LIN {X 0,Y 117.45,Z 837.122,A -85,B 0,C 180,E1 28506.231,E2 28506.231} C_VEL
LIN {X 0,Y 123.692,Z 839.313,A -85,B 0,C 180,E1 28517.447,E2 28517.447} C_VEL
LIN {X 0,Y 126.068,Z 840.042,A -85,B 0,C 180,E1 28523.129,E2 28523.129} C_VEL
LIN {X 0,Y 128.758,Z 840.316,A -85,B 0,C 180,E1 28530.003,E2 28530.003} C_VEL
LIN {X 0,Y 126.025,Z 840.042,A -85,B 0,C 180,E1 28536.88,E2 28536.88} C_VEL
LIN {X 0,Y 122.693,Z 839.07,A -85,B 0,C 180,E1 28544.243,E2 28544.243} C_VEL
LIN {X 0,Y 118.511,Z 837.415,A -85,B 0,C 180,E1 28552.461,E2 28552.461} C_VEL
LIN {X 0,Y 109.257,Z 835.091,A -85,B 0,C 180,E1 28564.022,E2 28564.022} C_VEL
LIN {X 0,Y 99.295,Z 832.926,A -85,B 0,C 180,E1 28577.915,E2 28577.915} C_VEL
LIN {X 0,Y 67.915,Z 840.094,A -85,B 0,C 180,E1 28563.751,E2 28563.751} C_VEL
LIN {X 0,Y 48.693,Z 842.803,A -85,B 0,C 180,E1 28530.008,E2 28530.008} C_VEL
LIN {X 0,Y 67.859,Z 840.097,A -85,B 0,C 180,E1 28496.232,E2 28496.232} C_VEL
LIN {X 0,Y 93.632,Z 834.401,A -85,B 0,C 180,E1 28483.517,E2 28483.517} C_VEL
LIN {X 0,Y 99.85,Z 833.009,A -85,B 0,C 180,E1 28482.861,E2 28482.861} C_VEL
LIN {X 0,Y 109.786,Z 835.227,A -85,B 0,C 180,E1 28496.651,E2 28496.651} C_VEL
LIN {X 0,Y 117.45,Z 837.122,A -85,B 0,C 180,E1 28506.231,E2 28506.231} C_VEL
LIN {X 0,Y 119.061,Z 838.09,A -85,B 0,C 180,E1 28510.313,E2 28510.313} C_VEL
LIN {X 0,Y 117.917,Z 840.331,A -85,B 0,C 180,E1 28523.404,E2 28523.404} C_VEL
LIN {X 0,Y 120.645,Z 840.568,A -85,B 0,C 180,E1 28530.003,E2 28530.003} C_VEL
LIN {X 0,Y 117.661,Z 840.304,A -85,B 0,C 180,E1 28537.372,E2 28537.372} C_VEL
LIN {X 0,Y 111.816,Z 838.693,A -85,B 0,C 180,E1 28549.125,E2 28549.125} C_VEL
LIN {X 0,Y 107.871,Z 837.778,A -85,B 0,C 180,E1 28554.818,E2 28554.818} C_VEL
LIN {X 0,Y 95.953,Z 835.393,A -85,B 0,C 180,E1 28570.441,E2 28570.441} C_VEL
LIN {X 0,Y 92.882,Z 835.886,A -85,B 0,C 180,E1 28570.537,E2 28570.537} C_VEL
LIN {X 0,Y 63.467,Z 841.732,A -85,B 0,C 180,E1 28547.957,E2 28547.957} C_VEL
LIN {X 0,Y 56.707,Z 842.554,A -85,B 0,C 180,E1 28530.007,E2 28530.007} C_VEL
LIN {X 0,Y 74.763,Z 839.843,A -85,B 0,C 180,E1 28499.702,E2 28499.702} C_VEL
LIN {X 0,Y 92.876,Z 835.889,A -85,B 0,C 180,E1 28489.471,E2 28489.471} C_VEL
LIN {X 0,Y 95.998,Z 835.377,A -85,B 0,C 180,E1 28489.529,E2 28489.529} C_VEL
LIN {X 0,Y 107.958,Z 837.777,A -85,B 0,C 180,E1 28505.212,E2 28505.212} C_VEL
LIN {X 0,Y 111.852,Z 838.68,A -85,B 0,C 180,E1 28510.823,E2 28510.823} C_VEL
LIN {X 0,Y 117.917,Z 840.331,A -85,B 0,C 180,E1 28523.404,E2 28523.404} C_VEL
LIN {X 0,Y 116.337,Z 840.614,A -85,B 0,C 180,E1 28527.551,E2 28527.551} C_VEL
LIN {X 0,Y 110.179,Z 840.674,A -85,B 0,C 180,E1 28534.68,E2 28534.68} C_VEL
LIN {X 0,Y 107.551,Z 840.278,A -85,B 0,C 180,E1 28540.803,E2 28540.803} C_VEL
LIN {X 0,Y 104.839,Z 839.648,A -85,B 0,C 180,E1 28546.735,E2 28546.735} C_VEL
LIN {X 0,Y 96.704,Z 838.168,A -85,B 0,C 180,E1 28557.918,E2 28557.918} C_VEL
LIN {X 0,Y 92.654,Z 837.576,A -85,B 0,C 180,E1 28562.71,E2 28562.71} C_VEL
LIN {X 0,Y 89.467,Z 838.001,A -85,B 0,C 180,E1 28562.489,E2 28562.489} C_VEL
LIN {X 0,Y 69.132,Z 841.835,A -85,B 0,C 180,E1 28542.614,E2 28542.614} C_VEL
LIN {X 0,Y 64.726,Z 842.305,A -85,B 0,C 180,E1 28530.006,E2 28530.006} C_VEL
LIN {X 0,Y 81.92,Z 839.588,A -85,B 0,C 180,E1 28502.585,E2 28502.585} C_VEL
LIN {X 0,Y 89.524,Z 837.982,A -85,B 0,C 180,E1 28497.454,E2 28497.454} C_VEL
LIN {X 0,Y 92.693,Z 837.57,A -85,B 0,C 180,E1 28497.288,E2 28497.288} C_VEL
LIN {X 0,Y 99.504,Z 838.587,A -85,B 0,C 180,E1 28505.514,E2 28505.514} C_VEL
LIN {X 0,Y 104.9,Z 839.648,A -85,B 0,C 180,E1 28513.283,E2 28513.283} C_VEL
LIN {X 0,Y 109.758,Z 840.638,A -85,B 0,C 180,E1 28524.137,E2 28524.137} C_VEL
LIN {X 0,Y 112.484,Z 840.821,A -85,B 0,C 180,E1 28530.004,E2 28530.004} C_VEL
LIN {X 0,Y 110.179,Z 840.674,A -85,B 0,C 180,E1 28534.68,E2 28534.68} C_VEL
LIN {X 0,Y 105.682,Z 840.634,A -85,B 0,C 180,E1 28538.598,E2 28538.598} C_VEL
LIN {X 0,Y 96.395,Z 840.259,A -85,B 0,C 180,E1 28545.328,E2 28545.328} C_VEL
LIN {X 0,Y 90.521,Z 839.276,A -85,B 0,C 180,E1 28554.711,E2 28554.711} C_VEL
LIN {X 0,Y 84.585,Z 840.315,A -85,B 0,C 180,E1 28550.909,E2 28550.909} C_VEL
LIN {X 0,Y 72.751,Z 842.055,A -85,B 0,C 180,E1 28530.006,E2 28530.006} C_VEL
LIN {X 0,Y 84.537,Z 840.318,A -85,B 0,C 180,E1 28509.089,E2 28509.089} C_VEL
LIN {X 0,Y 90.571,Z 839.27,A -85,B 0,C 180,E1 28505.276,E2 28505.276} C_VEL
LIN {X 0,Y 95.229,Z 840.033,A -85,B 0,C 180,E1 28511.974,E2 28511.974} C_VEL
LIN {X 0,Y 100.503,Z 840.844,A -85,B 0,C 180,E1 28521.369,E2 28521.369} C_VEL
LIN {X 0,Y 104.257,Z 841.077,A -85,B 0,C 180,E1 28530.004,E2 28530.004} C_VEL
LIN {X 0,Y 100.458,Z 840.844,A -85,B 0,C 180,E1 28538.643,E2 28538.643} C_VEL
LIN {X 0,Y 96.395,Z 840.259,A -85,B 0,C 180,E1 28545.328,E2 28545.328} C_VEL
LIN {X 0,Y 92.31,Z 840.489,A -85,B 0,C 180,E1 28545.322,E2 28545.322} C_VEL
LIN {X 0,Y 86.505,Z 841.177,A -85,B 0,C 180,E1 28541.158,E2 28541.158} C_VEL
LIN {X 0,Y 81.835,Z 841.654,A -85,B 0,C 180,E1 28533.397,E2 28533.397} C_VEL
LIN {X 0,Y 80.762,Z 841.807,A -85,B 0,C 180,E1 28530.005,E2 28530.005} C_VEL
LIN {X 0,Y 88.556,Z 840.741,A -85,B 0,C 180,E1 28515.404,E2 28515.404} C_VEL
LIN {X 0,Y 91.692,Z 841.15,A -85,B 0,C 180,E1 28520.966,E2 28520.966} C_VEL
LIN {X 0,Y 95.951,Z 841.335,A -85,B 0,C 180,E1 28530.004,E2 28530.004} C_VEL
LIN {X 0,Y 91.361,Z 841.131,A -85,B 0,C 180,E1 28539.512,E2 28539.512} C_VEL
LIN {X 0,Y 88.558,Z 840.746,A -85,B 0,C 180,E1 28544.541,E2 28544.541} C_VEL
LIN {X 0,Y 81.835,Z 841.654,A -85,B 0,C 180,E1 28533.397,E2 28533.397} C_VEL
LIN {X 0,Y 81.379,Z 843.653,A -85,B 0,C 180,E1 28532.075,E2 28532.075} C_VEL
LIN {X 0,Y 81.379,Z 862.5,A -85,B 0,C 180,E1 28532.075,E2 28532.075} C_VEL
LIN {X 0,Y 81.379,Z 862.5,A -85,B 0,C 180,E1 28532.075,E2 28532.075}

QRS_NEXT_CUT()
PTP {E1 28616.872,E2 28616.872}
PTP {X 0,Y 607.922,A -85,B 0,C 180,E1 28616.872,E2 28616.872,E3 0,E4 0,E5 0,E6 0}
QRS_SPEED_INIT()
LIN {X 0,Y 607.922,Z 862.5,A -85,B 0,C 180,E1 28616.872,E2 28616.872,E3 0,E4 0,E5 0,E6 0} C_VEL
LIN {X 0,Y 607.922,Z 274.59,A -85,B 0,C 180,E1 28616.872,E2 28616.872} C_VEL
LIN {X 0,Y 607.922,Z 266.51,A -85,B 0,C 180,E1 28616.872,E2 28616.872} C_VEL
LIN {X 0,Y 607.915,Z 264.51,A -85,B 0,C 180,E1 28616.683,E2 28616.683} C_VEL
LIN {X 0,Y 607.865,Z 264.511,A -85,B 0,C 180,E1 28613.578,E2 28613.578} C_VEL
LIN {X 0,Y 607.916,Z 264.507,A -85,B 0,C 180,E1 28610.438,E2 28610.438} C_VEL
LIN {X 0,Y 607.87,Z 264.512,A -85,B 0,C 180,E1 28607.363,E2 28607.363} C_VEL
LIN {X 0,Y 607.908,Z 264.506,A -85,B 0,C 180,E1 28604.155,E2 28604.155} C_VEL
LIN {X 0,Y 607.891,Z 264.513,A -85,B 0,C 180,E1 28600.994,E2 28600.994} C_VEL
LIN {X 0,Y 607.884,Z 264.508,A -85,B 0,C 180,E1 28597.771,E2 28597.771} C_VEL
LIN {X 0,Y 607.913,Z 264.516,A -85,B 0,C 180,E1 28594.683,E2 28594.683} C_VEL
LIN {X 0,Y 607.876,Z 264.509,A -85,B 0,C 180,E1 28591.44,E2 28591.44} C_VEL
LIN {X 0,Y 607.911,Z 264.511,A -85,B 0,C 180,E1 28588.354,E2 28588.354} C_VEL
LIN {X 0,Y 607.877,Z 264.509,A -85,B 0,C 180,E1 28585.312,E2 28585.312} C_VEL
LIN {X 0,Y 607.909,Z 264.511,A -85,B 0,C 180,E1 28582.277,E2 28582.277} C_VEL
LIN {X 0,Y 607.879,Z 264.51,A -85,B 0,C 180,E1 28579.165,E2 28579.165} C_VEL
LIN {X 0,Y 607.908,Z 264.508,A -85,B 0,C 180,E1 28576.046,E2 28576.046} C_VEL
LIN {X 0,Y 607.884,Z 264.511,A -85,B 0,C 180,E1 28572.917,E2 28572.917} C_VEL
LIN {X 0,Y 607.913,Z 264.506,A -85,B 0,C 180,E1 28569.776,E2 28569.776} C_VEL
LIN {X 0,Y 607.904,Z 264.514,A -85,B 0,C 180,E1 28566.54,E2 28566.54} C_VEL
LIN {X 0,Y 607.898,Z 264.506,A -85,B 0,C 180,E1 28563.322,E2 28563.322} C_VEL
LIN {X 0,Y 607.908,Z 264.512,A -85,B 0,C 180,E1 28560.102,E2 28560.102} C_VEL
LIN {X 0,Y 607.888,Z 264.508,A -85,B 0,C 180,E1 28556.94,E2 28556.94} C_VEL
LIN {X 0,Y 607.903,Z 264.508,A -85,B 0,C 180,E1 28553.763,E2 28553.763} C_VEL
LIN {X 0,Y 607.892,Z 264.511,A -85,B 0,C 180,E1 28550.628,E2 28550.628} C_VEL
LIN {X 0,Y 607.911,Z 264.505,A -85,B 0,C 180,E1 28547.418,E2 28547.418} C_VEL
LIN {X 0,Y 607.915,Z 264.514,A -85,B 0,C 180,E1 28544.088,E2 28544.088} C_VEL
LIN {X 0,Y 607.899,Z 264.506,A -85,B 0,C 180,E1 28540.903,E2 28540.903} C_VEL
LIN {X 0,Y 607.9,Z 264.511,A -85,B 0,C 180,E1 28537.751,E2 28537.751} C_VEL
LIN {X 0,Y 607.895,Z 264.508,A -85,B 0,C 180,E1 28534.623,E2 28534.623} C_VEL
LIN {X 0,Y 607.897,Z 264.509,A -85,B 0,C 180,E1 28531.508,E2 28531.508} C_VEL
LIN {X 0,Y 607.897,Z 264.51,A -85,B 0,C 180,E1 28528.398,E2 28528.398} C_VEL
LIN {X 0,Y 607.9,Z 264.506,A -85,B 0,C 180,E1 28525.188,E2 28525.188} C_VEL
LIN {X 0,Y 607.911,Z 264.515,A -85,B 0,C 180,E1 28521.944,E2 28521.944} C_VEL
LIN {X 0,Y 607.912,Z 264.505,A -85,B 0,C 180,E1 28518.713,E2 28518.713} C_VEL
LIN {X 0,Y 607.896,Z 264.512,A -85,B 0,C 180,E1 28515.522,E2 28515.522} C_VEL
LIN {X 0,Y 607.903,Z 264.508,A -85,B 0,C 180,E1 28512.384,E2 28512.384} C_VEL
LIN {X 0,Y 607.89,Z 264.51,A -85,B 0,C 180,E1 28509.291,E2 28509.291} C_VEL
LIN {X 0,Y 607.903,Z 264.508,A -85,B 0,C 180,E1 28506.237,E2 28506.237} C_VEL
LIN {X 0,Y 607.888,Z 264.508,A -85,B 0,C 180,E1 28503.06,E2 28503.06} C_VEL
LIN {X 0,Y 607.908,Z 264.512,A -85,B 0,C 180,E1 28499.892,E2 28499.892} C_VEL
LIN {X 0,Y 607.899,Z 264.506,A -85,B 0,C 180,E1 28496.673,E2 28496.673} C_VEL
LIN {X 0,Y 607.895,Z 264.512,A -85,B 0,C 180,E1 28493.342,E2 28493.342} C_VEL
LIN {X 0,Y 607.911,Z 264.506,A -85,B 0,C 180,E1 28490.183,E2 28490.183} C_VEL
LIN {X 0,Y 607.883,Z 264.511,A -85,B 0,C 180,E1 28487.049,E2 28487.049} C_VEL
LIN {X 0,Y 607.908,Z 264.509,A -85,B 0,C 180,E1 28483.914,E2 28483.914} C_VEL
LIN {X 0,Y 607.88,Z 264.509,A -85,B 0,C 180,E1 28480.768,E2 28480.768} C_VEL
LIN {X 0,Y 607.911,Z 264.513,A -85,B 0,C 180,E1 28477.604,E2 28477.604} C_VEL
LIN {X 0,Y 607.885,Z 264.508,A -85,B 0,C 180,E1 28474.459,E2 28474.459} C_VEL
LIN {X 0,Y 607.9,Z 264.514,A -85,B 0,C 180,E1 28471.205,E2 28471.205} C_VEL
LIN {X 0,Y 607.913,Z 264.506,A -85,B 0,C 180,E1 28467.969,E2 28467.969} C_VEL
LIN {X 0,Y 607.875,Z 264.511,A -85,B 0,C 180,E1 28464.78,E2 28464.78} C_VEL
LIN {X 0,Y 607.913,Z 264.508,A -85,B 0,C 180,E1 28461.682,E2 28461.682} C_VEL
LIN {X 0,Y 607.871,Z 264.511,A -85,B 0,C 180,E1 28458.609,E2 28458.609} C_VEL
LIN {X 0,Y 607.913,Z 264.509,A -85,B 0,C 180,E1 28455.551,E2 28455.551} C_VEL
LIN {X 0,Y 607.867,Z 264.511,A -85,B 0,C 180,E1 28452.443,E2 28452.443} C_VEL
LIN {X 0,Y 607.916,Z 264.512,A -85,B 0,C 180,E1 28449.276,E2 28449.276} C_VEL
LIN {X 0,Y 607.866,Z 264.51,A -85,B 0,C 180,E1 28446.232,E2 28446.232} C_VEL
LIN {X 0,Y 607.907,Z 264.515,A -85,B 0,C 180,E1 28443.017,E2 28443.017} C_VEL
LIN {X 0,Y 607.869,Z 264.51,A -85,B 0,C 180,E1 28440,E2 28440} C_VEL
LIN {X 0,Y 607.884,Z 264.513,A -85,B 0,C 180,E1 28436.734,E2 28436.734} C_VEL
LIN {X 0,Y 607.885,Z 264.509,A -85,B 0,C 180,E1 28433.673,E2 28433.673} C_VEL
LIN {X 0,Y 607.865,Z 264.512,A -85,B 0,C 180,E1 28430.437,E2 28430.437} C_VEL
LIN {X 0,Y 607.894,Z 264.509,A -85,B 0,C 180,E1 28427.461,E2 28427.461} C_VEL
LIN {X 0,Y 607.858,Z 264.512,A -85,B 0,C 180,E1 28424.252,E2 28424.252} C_VEL
LIN {X 0,Y 607.91,Z 264.51,A -85,B 0,C 180,E1 28421.194,E2 28421.194} C_VEL
LIN {X 0,Y 607.852,Z 264.512,A -85,B 0,C 180,E1 28418.075,E2 28418.075} C_VEL
LIN {X 0,Y 607.917,Z 264.509,A -85,B 0,C 180,E1 28415.099,E2 28415.099} C_VEL
LIN {X 0,Y 607.85,Z 264.513,A -85,B 0,C 180,E1 28412.042,E2 28412.042} C_VEL
LIN {X 0,Y 607.911,Z 264.51,A -85,B 0,C 180,E1 28409.016,E2 28409.016} C_VEL
LIN {X 0,Y 607.846,Z 264.513,A -85,B 0,C 180,E1 28405.881,E2 28405.881} C_VEL
LIN {X 0,Y 607.918,Z 264.511,A -85,B 0,C 180,E1 28402.871,E2 28402.871} C_VEL
LIN {X 0,Y 607.843,Z 264.513,A -85,B 0,C 180,E1 28399.849,E2 28399.849} C_VEL
LIN {X 0,Y 607.911,Z 264.511,A -85,B 0,C 180,E1 28396.826,E2 28396.826} C_VEL
LIN {X 0,Y 607.84,Z 264.514,A -85,B 0,C 180,E1 28393.77,E2 28393.77} C_VEL
LIN {X 0,Y 607.895,Z 264.511,A -85,B 0,C 180,E1 28390.835,E2 28390.835} C_VEL
LIN {X 0,Y 607.837,Z 264.508,A -85,B 0,C 180,E1 28387.701,E2 28387.701} C_VEL
LIN {X 0,Y 607.907,Z 264.795,A -85,B 0,C 180,E1 28386.686,E2 28386.686} C_VEL
LIN {X 0,Y 607.896,Z 291.162,A -85,B 0,C 180,E1 28383.838,E2 28383.838} C_VEL
LIN {X 0,Y 607.911,Z 305.952,A -85,B 0,C 180,E1 28382.324,E2 28382.324} C_VEL
LIN {X 0,Y 607.909,Z 526.839,A -85,B 0,C 180,E1 28379.341,E2 28379.341} C_VEL
LIN {X 0,Y 607.905,Z 607.712,A -85,B 0,C 180,E1 28378.247,E2 28378.247} C_VEL
LIN {X 0,Y 607.907,Z 629.078,A -85,B 0,C 180,E1 28377.784,E2 28377.784} C_VEL
LIN {X 0,Y 607.905,Z 650.472,A -85,B 0,C 180,E1 28377.15,E2 28377.15} C_VEL
LIN {X 0,Y 607.91,Z 670.867,A -85,B 0,C 180,E1 28376.364,E2 28376.364} C_VEL
LIN {X 0,Y 607.918,Z 690.753,A -85,B 0,C 180,E1 28375.421,E2 28375.421} C_VEL
LIN {X 0,Y 607.916,Z 710.113,A -85,B 0,C 180,E1 28374.331,E2 28374.331} C_VEL
LIN {X 0,Y 607.913,Z 729.302,A -85,B 0,C 180,E1 28373.044,E2 28373.044} C_VEL
LIN {X 0,Y 607.911,Z 746.772,A -85,B 0,C 180,E1 28371.677,E2 28371.677} C_VEL
LIN {X 0,Y 607.913,Z 763.659,A -85,B 0,C 180,E1 28370.155,E2 28370.155} C_VEL
LIN {X 0,Y 607.918,Z 779.471,A -85,B 0,C 180,E1 28368.507,E2 28368.507} C_VEL
LIN {X 0,Y 607.91,Z 794.115,A -85,B 0,C 180,E1 28366.728,E2 28366.728} C_VEL
LIN {X 0,Y 607.911,Z 806.544,A -85,B 0,C 180,E1 28364.964,E2 28364.964} C_VEL
LIN {X 0,Y 607.916,Z 817.733,A -85,B 0,C 180,E1 28363.119,E2 28363.119} C_VEL
LIN {X 0,Y 607.912,Z 827.063,A -85,B 0,C 180,E1 28361.287,E2 28361.287} C_VEL
LIN {X 0,Y 607.911,Z 835.464,A -85,B 0,C 180,E1 28359.275,E2 28359.275} C_VEL
LIN {X 0,Y 607.91,Z 842.128,A -85,B 0,C 180,E1 28357.276,E2 28357.276} C_VEL
LIN {X 0,Y 607.912,Z 847.015,A -85,B 0,C 180,E1 28355.285,E2 28355.285} C_VEL
LIN {X 0,Y 607.917,Z 850.447,A -85,B 0,C 180,E1 28353.206,E2 28353.206} C_VEL
LIN {X 0,Y 607.91,Z 852.21,A -85,B 0,C 180,E1 28351.225,E2 28351.225} C_VEL
LIN {X 0,Y 607.902,Z 852.329,A -85,B 0,C 180,E1 28349.246,E2 28349.246} C_VEL
LIN {X 0,Y 607.908,Z 850.896,A -85,B 0,C 180,E1 28347.172,E2 28347.172} C_VEL
LIN {X 0,Y 607.912,Z 847.987,A -85,B 0,C 180,E1 28345.188,E2 28345.188} C_VEL
LIN {X 0,Y 607.915,Z 843.399,A -85,B 0,C 180,E1 28343.199,E2 28343.199} C_VEL
LIN {X 0,Y 607.906,Z 837.238,A -85,B 0,C 180,E1 28341.202,E2 28341.202} C_VEL
LIN {X 0,Y 607.899,Z 829.658,A -85,B 0,C 180,E1 28339.289,E2 28339.289} C_VEL
LIN {X 0,Y 607.899,Z 820.329,A -85,B 0,C 180,E1 28337.364,E2 28337.364} C_VEL
LIN {X 0,Y 607.904,Z 809.746,A -85,B 0,C 180,E1 28335.523,E2 28335.523} C_VEL
LIN {X 0,Y 607.911,Z 797.742,A -85,B 0,C 180,E1 28333.764,E2 28333.764} C_VEL
LIN {X 0,Y 607.906,Z 783.722,A -85,B 0,C 180,E1 28331.989,E2 28331.989} C_VEL
LIN {X 0,Y 607.908,Z 768.722,A -85,B 0,C 180,E1 28330.346,E2 28330.346} C_VEL
LIN {X 0,Y 607.916,Z 751.704,A -85,B 0,C 180,E1 28328.737,E2 28328.737} C_VEL
LIN {X 0,Y 607.916,Z 733.47,A -85,B 0,C 180,E1 28327.263,E2 28327.263} C_VEL
LIN {X 0,Y 607.915,Z 714.947,A -85,B 0,C 180,E1 28325.98,E2 28325.98} C_VEL
LIN {X 0,Y 607.918,Z 695.722,A -85,B 0,C 180,E1 28324.84,E2 28324.84} C_VEL
LIN {X 0,Y 607.901,Z 676.877,A -85,B 0,C 180,E1 28323.902,E2 28323.902} C_VEL
LIN {X 0,Y 607.905,Z 656.219,A -85,B 0,C 180,E1 28323.057,E2 28323.057} C_VEL
LIN {X 0,Y 607.916,Z 636.206,A -85,B 0,C 180,E1 28322.402,E2 28322.402} C_VEL
LIN {X 0,Y 607.902,Z 616.001,A -85,B 0,C 180,E1 28321.914,E2 28321.914} C_VEL
LIN {X 0,Y 607.912,Z 593.483,A -85,B 0,C 180,E1 28321.54,E2 28321.54} C_VEL
LIN {X 0,Y 607.908,Z 369.551,A -85,B 0,C 180,E1 28318.548,E2 28318.548} C_VEL
LIN {X 0,Y 607.913,Z 305.698,A -85,B 0,C 180,E1 28317.66,E2 28317.66} C_VEL
LIN {X 0,Y 607.917,Z 279.428,A -85,B 0,C 180,E1 28314.913,E2 28314.913} C_VEL
LIN {X 0,Y 607.9,Z 264.617,A -85,B 0,C 180,E1 28313.27,E2 28313.27} C_VEL
LIN {X 0,Y 607.837,Z 264.514,A -85,B 0,C 180,E1 28310.339,E2 28310.339} C_VEL
LIN {X 0,Y 607.912,Z 264.514,A -85,B 0,C 180,E1 28307.324,E2 28307.324} C_VEL
LIN {X 0,Y 607.84,Z 264.512,A -85,B 0,C 180,E1 28304.314,E2 28304.314} C_VEL
LIN {X 0,Y 607.916,Z 264.513,A -85,B 0,C 180,E1 28301.264,E2 28301.264} C_VEL
LIN {X 0,Y 607.843,Z 264.511,A -85,B 0,C 180,E1 28298.206,E2 28298.206} C_VEL
LIN {X 0,Y 607.918,Z 264.511,A -85,B 0,C 180,E1 28295.145,E2 28295.145} C_VEL
LIN {X 0,Y 607.847,Z 264.513,A -85,B 0,C 180,E1 28292.094,E2 28292.094} C_VEL
LIN {X 0,Y 607.914,Z 264.511,A -85,B 0,C 180,E1 28289.025,E2 28289.025} C_VEL
LIN {X 0,Y 607.849,Z 264.512,A -85,B 0,C 180,E1 28286.052,E2 28286.052} C_VEL
LIN {X 0,Y 607.918,Z 264.512,A -85,B 0,C 180,E1 28283.044,E2 28283.044} C_VEL
LIN {X 0,Y 607.852,Z 264.511,A -85,B 0,C 180,E1 28280.007,E2 28280.007} C_VEL
LIN {X 0,Y 607.917,Z 264.511,A -85,B 0,C 180,E1 28276.925,E2 28276.925} C_VEL
LIN {X 0,Y 607.855,Z 264.511,A -85,B 0,C 180,E1 28273.896,E2 28273.896} C_VEL
LIN {X 0,Y 607.916,Z 264.51,A -85,B 0,C 180,E1 28270.807,E2 28270.807} C_VEL
LIN {X 0,Y 607.859,Z 264.511,A -85,B 0,C 180,E1 28267.752,E2 28267.752} C_VEL
LIN {X 0,Y 607.917,Z 264.508,A -85,B 0,C 180,E1 28264.623,E2 28264.623} C_VEL
LIN {X 0,Y 607.863,Z 264.511,A -85,B 0,C 180,E1 28261.602,E2 28261.602} C_VEL
LIN {X 0,Y 607.917,Z 264.507,A -85,B 0,C 180,E1 28258.492,E2 28258.492} C_VEL
LIN {X 0,Y 607.915,Z 264.51,A -85,B 0,C 180,E1 28256.683,E2 28256.683} C_VEL
LIN {X 0,Y 606.907,Z 264.632,A -85,B 0,C 180,E1 28255.957,E2 28255.957} C_VEL
LIN {X 0,Y 600.448,Z 265.435,A -85,B 0,C 180,E1 28253.921,E2 28253.921} C_VEL
LIN {X 0,Y 599.932,Z 265.501,A -85,B 0,C 180,E1 28253.391,E2 28253.391} C_VEL
LIN {X 0,Y 599.963,Z 265.495,A -85,B 0,C 180,E1 28250.213,E2 28250.213} C_VEL
LIN {X 0,Y 599.948,Z 265.502,A -85,B 0,C 180,E1 28247.096,E2 28247.096} C_VEL
LIN {X 0,Y 599.941,Z 265.496,A -85,B 0,C 180,E1 28243.84,E2 28243.84} C_VEL
LIN {X 0,Y 599.972,Z 265.505,A -85,B 0,C 180,E1 28240.733,E2 28240.733} C_VEL
LIN {X 0,Y 599.935,Z 265.498,A -85,B 0,C 180,E1 28237.564,E2 28237.564} C_VEL
LIN {X 0,Y 599.973,Z 265.5,A -85,B 0,C 180,E1 28234.429,E2 28234.429} C_VEL
LIN {X 0,Y 599.938,Z 265.5,A -85,B 0,C 180,E1 28231.236,E2 28231.236} C_VEL
LIN {X 0,Y 599.975,Z 265.496,A -85,B 0,C 180,E1 28228.111,E2 28228.111} C_VEL
LIN {X 0,Y 599.949,Z 265.502,A -85,B 0,C 180,E1 28224.903,E2 28224.903} C_VEL
LIN {X 0,Y 599.952,Z 265.496,A -85,B 0,C 180,E1 28221.56,E2 28221.56} C_VEL
LIN {X 0,Y 599.972,Z 265.504,A -85,B 0,C 180,E1 28218.438,E2 28218.438} C_VEL
LIN {X 0,Y 599.944,Z 265.498,A -85,B 0,C 180,E1 28215.231,E2 28215.231} C_VEL
LIN {X 0,Y 599.968,Z 265.5,A -85,B 0,C 180,E1 28212.132,E2 28212.132} C_VEL
LIN {X 0,Y 599.945,Z 265.498,A -85,B 0,C 180,E1 28209.046,E2 28209.046} C_VEL
LIN {X 0,Y 599.967,Z 265.497,A -85,B 0,C 180,E1 28205.911,E2 28205.911} C_VEL
LIN {X 0,Y 599.949,Z 265.5,A -85,B 0,C 180,E1 28202.794,E2 28202.794} C_VEL
LIN {X 0,Y 599.978,Z 265.493,A -85,B 0,C 180,E1 28199.552,E2 28199.552} C_VEL
LIN {X 0,Y 599.976,Z 265.503,A -85,B 0,C 180,E1 28196.207,E2 28196.207} C_VEL
LIN {X 0,Y 599.952,Z 265.497,A -85,B 0,C 180,E1 28192.952,E2 28192.952} C_VEL
LIN {X 0,Y 599.964,Z 265.5,A -85,B 0,C 180,E1 28189.875,E2 28189.875} C_VEL
LIN {X 0,Y 599.952,Z 265.498,A -85,B 0,C 180,E1 28186.757,E2 28186.757} C_VEL
LIN {X 0,Y 599.962,Z 265.497,A -85,B 0,C 180,E1 28183.59,E2 28183.59} C_VEL
LIN {X 0,Y 599.961,Z 265.501,A -85,B 0,C 180,E1 28180.369,E2 28180.369} C_VEL
LIN {X 0,Y 599.978,Z 265.493,A -85,B 0,C 180,E1 28177.084,E2 28177.084} C_VEL
LIN {X 0,Y 599.965,Z 265.501,A -85,B 0,C 180,E1 28173.822,E2 28173.822} C_VEL
LIN {X 0,Y 599.958,Z 265.497,A -85,B 0,C 180,E1 28170.573,E2 28170.573} C_VEL
LIN {X 0,Y 599.957,Z 265.498,A -85,B 0,C 180,E1 28167.421,E2 28167.421} C_VEL
LIN {X 0,Y 599.963,Z 265.501,A -85,B 0,C 180,E1 28164.221,E2 28164.221} C_VEL
LIN {X 0,Y 599.968,Z 265.494,A -85,B 0,C 180,E1 28160.988,E2 28160.988} C_VEL
LIN {X 0,Y 599.965,Z 265.502,A -85,B 0,C 180,E1 28157.684,E2 28157.684} C_VEL
LIN {X 0,Y 599.968,Z 265.495,A -85,B 0,C 180,E1 28154.536,E2 28154.536} C_VEL
LIN {X 0,Y 599.953,Z 265.499,A -85,B 0,C 180,E1 28151.339,E2 28151.339} C_VEL
LIN {X 0,Y 599.965,Z 265.499,A -85,B 0,C 180,E1 28148.164,E2 28148.164} C_VEL
LIN {X 0,Y 599.953,Z 265.496,A -85,B 0,C 180,E1 28144.957,E2 28144.957} C_VEL
LIN {X 0,Y 599.972,Z 265.504,A -85,B 0,C 180,E1 28141.753,E2 28141.753} C_VEL
LIN {X 0,Y 599.972,Z 265.494,A -85,B 0,C 180,E1 28138.448,E2 28138.448} C_VEL
LIN {X 0,Y 599.951,Z 265.5,A -85,B 0,C 180,E1 28135.247,E2 28135.247} C_VEL
LIN {X 0,Y 599.968,Z 265.497,A -85,B 0,C 180,E1 28132.053,E2 28132.053} C_VEL
LIN {X 0,Y 599.945,Z 265.498,A -85,B 0,C 180,E1 28128.876,E2 28128.876} C_VEL
LIN {X 0,Y 599.973,Z 265.503,A -85,B 0,C 180,E1 28125.637,E2 28125.637} C_VEL
LIN {X 0,Y 599.959,Z 265.495,A -85,B 0,C 180,E1 28122.417,E2 28122.417} C_VEL
LIN {X 0,Y 599.952,Z 265.502,A -85,B 0,C 180,E1 28119.17,E2 28119.17} C_VEL
LIN {X 0,Y 599.977,Z 265.495,A -85,B 0,C 180,E1 28116.034,E2 28116.034} C_VEL
LIN {X 0,Y 599.938,Z 265.5,A -85,B 0,C 180,E1 28112.796,E2 28112.796} C_VEL
LIN {X 0,Y 599.972,Z 265.499,A -85,B 0,C 180,E1 28109.667,E2 28109.667} C_VEL
LIN {X 0,Y 599.936,Z 265.498,A -85,B 0,C 180,E1 28106.529,E2 28106.529} C_VEL
LIN {X 0,Y 599.977,Z 265.504,A -85,B 0,C 180,E1 28103.334,E2 28103.334} C_VEL
LIN {X 0,Y 599.946,Z 265.497,A -85,B 0,C 180,E1 28100.181,E2 28100.181} C_VEL
LIN {X 0,Y 599.942,Z 265.5,A -85,B 0,C 180,E1 28096.857,E2 28096.857} C_VEL
LIN {X 0,Y 599.974,Z 265.496,A -85,B 0,C 180,E1 28093.688,E2 28093.688} C_VEL
LIN {X 0,Y 599.928,Z 265.498,A -85,B 0,C 180,E1 28090.491,E2 28090.491} C_VEL
LIN {X 0,Y 599.975,Z 265.499,A -85,B 0,C 180,E1 28087.373,E2 28087.373} C_VEL
LIN {X 0,Y 599.925,Z 265.498,A -85,B 0,C 180,E1 28084.301,E2 28084.301} C_VEL
LIN {X 0,Y 599.978,Z 265.502,A -85,B 0,C 180,E1 28081.146,E2 28081.146} C_VEL
LIN {X 0,Y 599.925,Z 265.498,A -85,B 0,C 180,E1 28078.09,E2 28078.09} C_VEL
LIN {X 0,Y 599.969,Z 265.504,A -85,B 0,C 180,E1 28074.933,E2 28074.933} C_VEL
LIN {X 0,Y 599.929,Z 265.498,A -85,B 0,C 180,E1 28071.856,E2 28071.856} C_VEL
LIN {X 0,Y 599.936,Z 265.503,A -85,B 0,C 180,E1 28068.561,E2 28068.561} C_VEL
LIN {X 0,Y 599.946,Z 265.497,A -85,B 0,C 180,E1 28065.523,E2 28065.523} C_VEL
LIN {X 0,Y 599.924,Z 265.502,A -85,B 0,C 180,E1 28062.342,E2 28062.342} C_VEL
LIN {X 0,Y 599.957,Z 265.497,A -85,B 0,C 180,E1 28059.31,E2 28059.31} C_VEL
LIN {X 0,Y 599.917,Z 265.502,A -85,B 0,C 180,E1 28056.201,E2 28056.201} C_VEL
LIN {X 0,Y 599.962,Z 265.498,A -85,B 0,C 180,E1 28053.152,E2 28053.152} C_VEL
LIN {X 0,Y 599.91,Z 265.501,A -85,B 0,C 180,E1 28050,E2 28050} C_VEL
LIN {X 0,Y 599.97,Z 265.501,A -85,B 0,C 180,E1 28046.954,E2 28046.954} C_VEL
LIN {X 0,Y 599.906,Z 265.502,A -85,B 0,C 180,E1 28043.843,E2 28043.843} C_VEL
LIN {X 0,Y 599.977,Z 265.499,A -85,B 0,C 180,E1 28040.709,E2 28040.709} C_VEL
LIN {X 0,Y 599.902,Z 265.502,A -85,B 0,C 180,E1 28037.674,E2 28037.674} C_VEL
LIN {X 0,Y 599.977,Z 265.501,A -85,B 0,C 180,E1 28034.636,E2 28034.636} C_VEL
LIN {X 0,Y 599.9,Z 265.5,A -85,B 0,C 180,E1 28031.552,E2 28031.552} C_VEL
LIN {X 0,Y 599.964,Z 265.49,A -85,B 0,C 180,E1 28028.433,E2 28028.433} C_VEL
LIN {X 0,Y 599.952,Z 265.771,A -85,B 0,C 180,E1 28027.148,E2 28027.148} C_VEL
LIN {X 0,Y 600.718,Z 268.698,A -85,B 0,C 180,E1 28026.752,E2 28026.752} C_VEL
LIN {X 0,Y 600.596,Z 297.234,A -85,B 0,C 180,E1 28023.655,E2 28023.655} C_VEL
LIN {X 0,Y 600.676,Z 306.011,A -85,B 0,C 180,E1 28022.76,E2 28022.76} C_VEL
LIN {X 0,Y 601.139,Z 309.101,A -85,B 0,C 180,E1 28022.684,E2 28022.684} C_VEL
LIN {X 0,Y 600.923,Z 532.92,A -85,B 0,C 180,E1 28019.635,E2 28019.635} C_VEL
LIN {X 0,Y 600.845,Z 608.42,A -85,B 0,C 180,E1 28018.597,E2 28018.597} C_VEL
LIN {X 0,Y 600.788,Z 630.03,A -85,B 0,C 180,E1 28018.118,E2 28018.118} C_VEL
LIN {X 0,Y 600.702,Z 651.095,A -85,B 0,C 180,E1 28017.481,E2 28017.481} C_VEL
LIN {X 0,Y 600.637,Z 671.573,A -85,B 0,C 180,E1 28016.679,E2 28016.679} C_VEL
LIN {X 0,Y 600.537,Z 691.746,A -85,B 0,C 180,E1 28015.703,E2 28015.703} C_VEL
LIN {X 0,Y 600.436,Z 710.943,A -85,B 0,C 180,E1 28014.601,E2 28014.601} C_VEL
LIN {X 0,Y 600.345,Z 730.759,A -85,B 0,C 180,E1 28013.248,E2 28013.248} C_VEL
LIN {X 0,Y 600.244,Z 748.692,A -85,B 0,C 180,E1 28011.805,E2 28011.805} C_VEL
LIN {X 0,Y 600.16,Z 765.688,A -85,B 0,C 180,E1 28010.223,E2 28010.223} C_VEL
LIN {X 0,Y 600.089,Z 781.24,A -85,B 0,C 180,E1 28008.548,E2 28008.548} C_VEL
LIN {X 0,Y 600.026,Z 795.618,A -85,B 0,C 180,E1 28006.755,E2 28006.755} C_VEL
LIN {X 0,Y 599.986,Z 807.828,A -85,B 0,C 180,E1 28004.969,E2 28004.969} C_VEL
LIN {X 0,Y 599.949,Z 819.294,A -85,B 0,C 180,E1 28003.002,E2 28003.002} C_VEL
LIN {X 0,Y 599.934,Z 828.846,A -85,B 0,C 180,E1 28001.049,E2 28001.049} C_VEL
LIN {X 0,Y 599.929,Z 836.53,A -85,B 0,C 180,E1 27999.11,E2 27999.11} C_VEL
LIN {X 0,Y 599.921,Z 843.146,A -85,B 0,C 180,E1 27996.988,E2 27996.988} C_VEL
LIN {X 0,Y 599.916,Z 847.823,A -85,B 0,C 180,E1 27994.972,E2 27994.972} C_VEL
LIN {X 0,Y 599.909,Z 850.899,A -85,B 0,C 180,E1 27992.866,E2 27992.866} C_VEL
LIN {X 0,Y 599.903,Z 852.329,A -85,B 0,C 180,E1 27990.764,E2 27990.764} C_VEL
LIN {X 0,Y 599.907,Z 852.209,A -85,B 0,C 180,E1 27988.759,E2 27988.759} C_VEL
LIN {X 0,Y 599.916,Z 850.337,A -85,B 0,C 180,E1 27986.656,E2 27986.656} C_VEL
LIN {X 0,Y 599.915,Z 846.812,A -85,B 0,C 180,E1 27984.549,E2 27984.549} C_VEL
LIN {X 0,Y 599.912,Z 841.873,A -85,B 0,C 180,E1 27982.531,E2 27982.531} C_VEL
LIN {X 0,Y 599.915,Z 835.111,A -85,B 0,C 180,E1 27980.503,E2 27980.503} C_VEL
LIN {X 0,Y 599.93,Z 826.604,A -85,B 0,C 180,E1 27978.464,E2 27978.464} C_VEL
LIN {X 0,Y 599.957,Z 816.689,A -85,B 0,C 180,E1 27976.508,E2 27976.508} C_VEL
LIN {X 0,Y 599.998,Z 805.263,A -85,B 0,C 180,E1 27974.636,E2 27974.636} C_VEL
LIN {X 0,Y 600.051,Z 791.452,A -85,B 0,C 180,E1 27972.704,E2 27972.704} C_VEL
LIN {X 0,Y 600.105,Z 776.746,A -85,B 0,C 180,E1 27970.94,E2 27970.94} C_VEL
LIN {X 0,Y 600.19,Z 760.551,A -85,B 0,C 180,E1 27969.268,E2 27969.268} C_VEL
LIN {X 0,Y 600.267,Z 743.47,A -85,B 0,C 180,E1 27967.75,E2 27967.75} C_VEL
LIN {X 0,Y 600.363,Z 725.061,A -85,B 0,C 180,E1 27966.345,E2 27966.345} C_VEL
LIN {X 0,Y 600.473,Z 705.754,A -85,B 0,C 180,E1 27965.086,E2 27965.086} C_VEL
LIN {X 0,Y 600.575,Z 685.751,A -85,B 0,C 180,E1 27963.981,E2 27963.981} C_VEL
LIN {X 0,Y 600.653,Z 665.781,A -85,B 0,C 180,E1 27963.079,E2 27963.079} C_VEL
LIN {X 0,Y 600.749,Z 643.921,A -85,B 0,C 180,E1 27962.284,E2 27962.284} C_VEL
LIN {X 0,Y 600.805,Z 622.361,A -85,B 0,C 180,E1 27961.687,E2 27961.687} C_VEL
LIN {X 0,Y 600.86,Z 602.046,A -85,B 0,C 180,E1 27961.302,E2 27961.302} C_VEL
LIN {X 0,Y 601.079,Z 368.915,A -85,B 0,C 180,E1 27958.14,E2 27958.14} C_VEL
LIN {X 0,Y 600.936,Z 307.014,A -85,B 0,C 180,E1 27957.274,E2 27957.274} C_VEL
LIN {X 0,Y 600.62,Z 305.582,A -85,B 0,C 180,E1 27957.212,E2 27957.212} C_VEL
LIN {X 0,Y 600.691,Z 275.467,A -85,B 0,C 180,E1 27953.994,E2 27953.994} C_VEL
LIN {X 0,Y 600.552,Z 267.725,A -85,B 0,C 180,E1 27953.128,E2 27953.128} C_VEL
LIN {X 0,Y 599.915,Z 265.554,A -85,B 0,C 180,E1 27952.785,E2 27952.785} C_VEL
LIN {X 0,Y 599.928,Z 265.505,A -85,B 0,C 180,E1 27949.837,E2 27949.837} C_VEL
LIN {X 0,Y 599.906,Z 265.503,A -85,B 0,C 180,E1 27946.608,E2 27946.608} C_VEL
LIN {X 0,Y 599.931,Z 265.501,A -85,B 0,C 180,E1 27943.761,E2 27943.761} C_VEL
LIN {X 0,Y 599.91,Z 265.501,A -85,B 0,C 180,E1 27940.537,E2 27940.537} C_VEL
LIN {X 0,Y 599.944,Z 265.499,A -85,B 0,C 180,E1 27937.587,E2 27937.587} C_VEL
LIN {X 0,Y 599.911,Z 265.501,A -85,B 0,C 180,E1 27934.402,E2 27934.402} C_VEL
LIN {X 0,Y 599.954,Z 265.504,A -85,B 0,C 180,E1 27931.433,E2 27931.433} C_VEL
LIN {X 0,Y 599.916,Z 265.501,A -85,B 0,C 180,E1 27928.359,E2 27928.359} C_VEL
LIN {X 0,Y 599.957,Z 265.502,A -85,B 0,C 180,E1 27925.36,E2 27925.36} C_VEL
LIN {X 0,Y 599.916,Z 265.5,A -85,B 0,C 180,E1 27922.23,E2 27922.23} C_VEL
LIN {X 0,Y 599.975,Z 265.502,A -85,B 0,C 180,E1 27919.166,E2 27919.166} C_VEL
LIN {X 0,Y 599.917,Z 265.499,A -85,B 0,C 180,E1 27916.061,E2 27916.061} C_VEL
LIN {X 0,Y 599.975,Z 265.503,A -85,B 0,C 180,E1 27913.002,E2 27913.002} C_VEL
LIN {X 0,Y 599.919,Z 265.499,A -85,B 0,C 180,E1 27909.885,E2 27909.885} C_VEL
LIN {X 0,Y 599.978,Z 265.5,A -85,B 0,C 180,E1 27906.795,E2 27906.795} C_VEL
LIN {X 0,Y 599.922,Z 265.499,A -85,B 0,C 180,E1 27903.727,E2 27903.727} C_VEL
LIN {X 0,Y 599.979,Z 265.497,A -85,B 0,C 180,E1 27900.573,E2 27900.573} C_VEL
LIN {X 0,Y 599.928,Z 265.5,A -85,B 0,C 180,E1 27897.516,E2 27897.516} C_VEL
LIN {X 0,Y 599.972,Z 265.496,A -85,B 0,C 180,E1 27894.357,E2 27894.357} C_VEL
LIN {X 0,Y 599.932,Z 265.501,A -85,B 0,C 180,E1 27893.391,E2 27893.391} C_VEL
LIN {X 0,Y 598.978,Z 265.626,A -85,B 0,C 180,E1 27892.655,E2 27892.655} C_VEL
LIN {X 0,Y 592.477,Z 266.431,A -85,B 0,C 180,E1 27890.538,E2 27890.538} C_VEL
LIN {X 0,Y 592.009,Z 266.483,A -85,B 0,C 180,E1 27890.054,E2 27890.054} C_VEL
LIN {X 0,Y 592.027,Z 266.492,A -85,B 0,C 180,E1 27886.92,E2 27886.92} C_VEL
LIN {X 0,Y 591.997,Z 266.485,A -85,B 0,C 180,E1 27883.718,E2 27883.718} C_VEL
LIN {X 0,Y 592.037,Z 266.49,A -85,B 0,C 180,E1 27880.567,E2 27880.567} C_VEL
LIN {X 0,Y 591.995,Z 266.489,A -85,B 0,C 180,E1 27877.351,E2 27877.351} C_VEL
LIN {X 0,Y 592.036,Z 266.485,A -85,B 0,C 180,E1 27874.169,E2 27874.169} C_VEL
LIN {X 0,Y 592.007,Z 266.491,A -85,B 0,C 180,E1 27871.006,E2 27871.006} C_VEL
LIN {X 0,Y 592.01,Z 266.486,A -85,B 0,C 180,E1 27867.63,E2 27867.63} C_VEL
LIN {X 0,Y 592.033,Z 266.492,A -85,B 0,C 180,E1 27864.482,E2 27864.482} C_VEL
LIN {X 0,Y 592.002,Z 266.487,A -85,B 0,C 180,E1 27861.285,E2 27861.285} C_VEL
LIN {X 0,Y 592.031,Z 266.488,A -85,B 0,C 180,E1 27858.139,E2 27858.139} C_VEL
LIN {X 0,Y 592.006,Z 266.489,A -85,B 0,C 180,E1 27854.955,E2 27854.955} C_VEL
LIN {X 0,Y 592.039,Z 266.483,A -85,B 0,C 180,E1 27851.712,E2 27851.712} C_VEL
LIN {X 0,Y 592.037,Z 266.493,A -85,B 0,C 180,E1 27848.407,E2 27848.407} C_VEL
LIN {X 0,Y 592.012,Z 266.486,A -85,B 0,C 180,E1 27845.163,E2 27845.163} C_VEL
LIN {X 0,Y 592.029,Z 266.488,A -85,B 0,C 180,E1 27842.025,E2 27842.025} C_VEL
LIN {X 0,Y 592.01,Z 266.487,A -85,B 0,C 180,E1 27838.883,E2 27838.883} C_VEL
LIN {X 0,Y 592.028,Z 266.485,A -85,B 0,C 180,E1 27835.723,E2 27835.723} C_VEL
LIN {X 0,Y 592.018,Z 266.49,A -85,B 0,C 180,E1 27832.508,E2 27832.508} C_VEL
LIN {X 0,Y 592.031,Z 266.483,A -85,B 0,C 180,E1 27829.227,E2 27829.227} C_VEL
LIN {X 0,Y 592.03,Z 266.491,A -85,B 0,C 180,E1 27825.979,E2 27825.979} C_VEL
LIN {X 0,Y 592.017,Z 266.486,A -85,B 0,C 180,E1 27822.782,E2 27822.782} C_VEL
LIN {X 0,Y 592.022,Z 266.487,A -85,B 0,C 180,E1 27819.625,E2 27819.625} C_VEL
LIN {X 0,Y 592.021,Z 266.489,A -85,B 0,C 180,E1 27816.4,E2 27816.4} C_VEL
LIN {X 0,Y 592.033,Z 266.483,A -85,B 0,C 180,E1 27813.098,E2 27813.098} C_VEL
LIN {X 0,Y 592.028,Z 266.491,A -85,B 0,C 180,E1 27809.806,E2 27809.806} C_VEL
LIN {X 0,Y 592.023,Z 266.485,A -85,B 0,C 180,E1 27806.611,E2 27806.611} C_VEL
LIN {X 0,Y 592.017,Z 266.487,A -85,B 0,C 180,E1 27803.405,E2 27803.405} C_VEL
LIN {X 0,Y 592.025,Z 266.49,A -85,B 0,C 180,E1 27800.179,E2 27800.179} C_VEL
LIN {X 0,Y 592.031,Z 266.483,A -85,B 0,C 180,E1 27796.921,E2 27796.921} C_VEL
LIN {X 0,Y 592.023,Z 266.491,A -85,B 0,C 180,E1 27793.594,E2 27793.594} C_VEL
LIN {X 0,Y 592.026,Z 266.486,A -85,B 0,C 180,E1 27790.362,E2 27790.362} C_VEL
LIN {X 0,Y 592.012,Z 266.488,A -85,B 0,C 180,E1 27787.242,E2 27787.242} C_VEL
LIN {X 0,Y 592.027,Z 266.488,A -85,B 0,C 180,E1 27784.062,E2 27784.062} C_VEL
LIN {X 0,Y 592.014,Z 266.485,A -85,B 0,C 180,E1 27780.896,E2 27780.896} C_VEL
LIN {X 0,Y 592.032,Z 266.493,A -85,B 0,C 180,E1 27777.611,E2 27777.611} C_VEL
LIN {X 0,Y 592.037,Z 266.483,A -85,B 0,C 180,E1 27774.324,E2 27774.324} C_VEL
LIN {X 0,Y 592.007,Z 266.489,A -85,B 0,C 180,E1 27771.078,E2 27771.078} C_VEL
LIN {X 0,Y 592.029,Z 266.488,A -85,B 0,C 180,E1 27767.897,E2 27767.897} C_VEL
LIN {X 0,Y 592.005,Z 266.487,A -85,B 0,C 180,E1 27764.772,E2 27764.772} C_VEL
LIN {X 0,Y 592.033,Z 266.493,A -85,B 0,C 180,E1 27761.57,E2 27761.57} C_VEL
LIN {X 0,Y 592.024,Z 266.484,A -85,B 0,C 180,E1 27758.303,E2 27758.303} C_VEL
LIN {X 0,Y 592.006,Z 266.49,A -85,B 0,C 180,E1 27755.004,E2 27755.004} C_VEL
LIN {X 0,Y 592.034,Z 266.487,A -85,B 0,C 180,E1 27751.798,E2 27751.798} C_VEL
LIN {X 0,Y 591.997,Z 266.488,A -85,B 0,C 180,E1 27748.663,E2 27748.663} C_VEL
LIN {X 0,Y 592.035,Z 266.49,A -85,B 0,C 180,E1 27745.509,E2 27745.509} C_VEL
LIN {X 0,Y 592.001,Z 266.487,A -85,B 0,C 180,E1 27742.334,E2 27742.334} C_VEL
LIN {X 0,Y 592.016,Z 266.492,A -85,B 0,C 180,E1 27739.024,E2 27739.024} C_VEL
LIN {X 0,Y 592.037,Z 266.482,A -85,B 0,C 180,E1 27735.778,E2 27735.778} C_VEL
LIN {X 0,Y 591.991,Z 266.49,A -85,B 0,C 180,E1 27732.584,E2 27732.584} C_VEL
LIN {X 0,Y 592.037,Z 266.485,A -85,B 0,C 180,E1 27729.429,E2 27729.429} C_VEL
LIN {X 0,Y 591.988,Z 266.488,A -85,B 0,C 180,E1 27726.303,E2 27726.303} C_VEL
LIN {X 0,Y 592.033,Z 266.489,A -85,B 0,C 180,E1 27723.098,E2 27723.098} C_VEL
LIN {X 0,Y 591.992,Z 266.488,A -85,B 0,C 180,E1 27720,E2 27720} C_VEL
LIN {X 0,Y 592.004,Z 266.49,A -85,B 0,C 180,E1 27716.708,E2 27716.708} C_VEL
LIN {X 0,Y 592.014,Z 266.487,A -85,B 0,C 180,E1 27713.6,E2 27713.6} C_VEL
LIN {X 0,Y 591.985,Z 266.489,A -85,B 0,C 180,E1 27710.374,E2 27710.374} C_VEL
LIN {X 0,Y 592.033,Z 266.487,A -85,B 0,C 180,E1 27707.317,E2 27707.317} C_VEL
LIN {X 0,Y 591.978,Z 266.489,A -85,B 0,C 180,E1 27704.12,E2 27704.12} C_VEL
LIN {X 0,Y 592.04,Z 266.491,A -85,B 0,C 180,E1 27700.977,E2 27700.977} C_VEL
LIN {X 0,Y 591.975,Z 266.489,A -85,B 0,C 180,E1 27697.874,E2 27697.874} C_VEL
LIN {X 0,Y 592.025,Z 266.49,A -85,B 0,C 180,E1 27694.705,E2 27694.705} C_VEL
LIN {X 0,Y 591.976,Z 266.49,A -85,B 0,C 180,E1 27691.666,E2 27691.666} C_VEL
LIN {X 0,Y 592,Z 266.493,A -85,B 0,C 180,E1 27688.428,E2 27688.428} C_VEL
LIN {X 0,Y 591.976,Z 266.489,A -85,B 0,C 180,E1 27685.509,E2 27685.509} C_VEL
LIN {X 0,Y 591.982,Z 266.486,A -85,B 0,C 180,E1 27682.186,E2 27682.186} C_VEL
LIN {X 0,Y 591.981,Z 266.49,A -85,B 0,C 180,E1 27679.311,E2 27679.311} C_VEL
LIN {X 0,Y 591.973,Z 266.489,A -85,B 0,C 180,E1 27676.014,E2 27676.014} C_VEL
LIN {X 0,Y 591.985,Z 266.492,A -85,B 0,C 180,E1 27673.144,E2 27673.144} C_VEL
LIN {X 0,Y 591.969,Z 266.494,A -85,B 0,C 180,E1 27669.927,E2 27669.927} C_VEL
LIN {X 0,Y 591.985,Z 266.677,A -85,B 0,C 180,E1 27667.64,E2 27667.64} C_VEL
LIN {X 0,Y 593.526,Z 271.971,A -85,B 0,C 180,E1 27666.903,E2 27666.903} C_VEL
LIN {X 0,Y 593.28,Z 300.35,A -85,B 0,C 180,E1 27663.789,E2 27663.789} C_VEL
LIN {X 0,Y 593.342,Z 305.975,A -85,B 0,C 180,E1 27663.22,E2 27663.22} C_VEL
LIN {X 0,Y 594.399,Z 310.515,A -85,B 0,C 180,E1 27663.082,E2 27663.082} C_VEL
LIN {X 0,Y 593.965,Z 533.81,A -85,B 0,C 180,E1 27660.005,E2 27660.005} C_VEL
LIN {X 0,Y 593.811,Z 608.503,A -85,B 0,C 180,E1 27658.966,E2 27658.966} C_VEL
LIN {X 0,Y 593.691,Z 630.401,A -85,B 0,C 180,E1 27658.476,E2 27658.476} C_VEL
LIN {X 0,Y 593.523,Z 651.814,A -85,B 0,C 180,E1 27657.815,E2 27657.815} C_VEL
LIN {X 0,Y 593.371,Z 673.436,A -85,B 0,C 180,E1 27656.952,E2 27656.952} C_VEL
LIN {X 0,Y 593.171,Z 692.742,A -85,B 0,C 180,E1 27655.992,E2 27655.992} C_VEL
LIN {X 0,Y 592.957,Z 712.555,A -85,B 0,C 180,E1 27654.826,E2 27654.826} C_VEL
LIN {X 0,Y 592.777,Z 731.677,A -85,B 0,C 180,E1 27653.491,E2 27653.491} C_VEL
LIN {X 0,Y 592.584,Z 749.296,A -85,B 0,C 180,E1 27652.05,E2 27652.05} C_VEL
LIN {X 0,Y 592.41,Z 766.197,A -85,B 0,C 180,E1 27650.448,E2 27650.448} C_VEL
LIN {X 0,Y 592.264,Z 782.03,A -85,B 0,C 180,E1 27648.708,E2 27648.708} C_VEL
LIN {X 0,Y 592.146,Z 796.325,A -85,B 0,C 180,E1 27646.883,E2 27646.883} C_VEL
LIN {X 0,Y 592.069,Z 808.47,A -85,B 0,C 180,E1 27645.074,E2 27645.074} C_VEL
LIN {X 0,Y 591.996,Z 819.817,A -85,B 0,C 180,E1 27643.08,E2 27643.08} C_VEL
LIN {X 0,Y 591.956,Z 829.331,A -85,B 0,C 180,E1 27641.083,E2 27641.083} C_VEL
LIN {X 0,Y 591.94,Z 836.886,A -85,B 0,C 180,E1 27639.136,E2 27639.136} C_VEL
LIN {X 0,Y 591.926,Z 843.147,A -85,B 0,C 180,E1 27637.083,E2 27637.083} C_VEL
LIN {X 0,Y 591.917,Z 847.819,A -85,B 0,C 180,E1 27635.039,E2 27635.039} C_VEL
LIN {X 0,Y 591.911,Z 850.902,A -85,B 0,C 180,E1 27632.905,E2 27632.905} C_VEL
LIN {X 0,Y 591.903,Z 852.329,A -85,B 0,C 180,E1 27630.774,E2 27630.774} C_VEL
LIN {X 0,Y 591.906,Z 852.208,A -85,B 0,C 180,E1 27628.742,E2 27628.742} C_VEL
LIN {X 0,Y 591.914,Z 850.34,A -85,B 0,C 180,E1 27626.611,E2 27626.611} C_VEL
LIN {X 0,Y 591.917,Z 846.814,A -85,B 0,C 180,E1 27624.475,E2 27624.475} C_VEL
LIN {X 0,Y 591.919,Z 841.873,A -85,B 0,C 180,E1 27622.429,E2 27622.429} C_VEL
LIN {X 0,Y 591.927,Z 835.112,A -85,B 0,C 180,E1 27620.374,E2 27620.374} C_VEL
LIN {X 0,Y 591.957,Z 826.608,A -85,B 0,C 180,E1 27618.306,E2 27618.306} C_VEL
LIN {X 0,Y 592.01,Z 816.685,A -85,B 0,C 180,E1 27616.323,E2 27616.323} C_VEL
LIN {X 0,Y 592.078,Z 805.264,A -85,B 0,C 180,E1 27614.425,E2 27614.425} C_VEL
LIN {X 0,Y 592.188,Z 791.79,A -85,B 0,C 180,E1 27612.511,E2 27612.511} C_VEL
LIN {X 0,Y 592.31,Z 777.679,A -85,B 0,C 180,E1 27610.782,E2 27610.782} C_VEL
LIN {X 0,Y 592.478,Z 761.096,A -85,B 0,C 180,E1 27609.037,E2 27609.037} C_VEL
LIN {X 0,Y 592.635,Z 743.864,A -85,B 0,C 180,E1 27607.482,E2 27607.482} C_VEL
LIN {X 0,Y 592.822,Z 725.868,A -85,B 0,C 180,E1 27606.084,E2 27606.084} C_VEL
LIN {X 0,Y 593.041,Z 706.649,A -85,B 0,C 180,E1 27604.805,E2 27604.805} C_VEL
LIN {X 0,Y 593.238,Z 686.778,A -85,B 0,C 180,E1 27603.688,E2 27603.688} C_VEL
LIN {X 0,Y 593.41,Z 666.487,A -85,B 0,C 180,E1 27602.753,E2 27602.753} C_VEL
LIN {X 0,Y 593.604,Z 644.936,A -85,B 0,C 180,E1 27601.953,E2 27601.953} C_VEL
LIN {X 0,Y 593.731,Z 622.882,A -85,B 0,C 180,E1 27601.331,E2 27601.331} C_VEL
LIN {X 0,Y 593.833,Z 602.403,A -85,B 0,C 180,E1 27600.936,E2 27600.936} C_VEL
LIN {X 0,Y 594.278,Z 370.188,A -85,B 0,C 180,E1 27597.75,E2 27597.75} C_VEL
LIN {X 0,Y 594.201,Z 308.915,A -85,B 0,C 180,E1 27596.883,E2 27596.883} C_VEL
LIN {X 0,Y 593.297,Z 305.655,A -85,B 0,C 180,E1 27596.759,E2 27596.759} C_VEL
LIN {X 0,Y 593.479,Z 277.228,A -85,B 0,C 180,E1 27593.683,E2 27593.683} C_VEL
LIN {X 0,Y 593.418,Z 271.187,A -85,B 0,C 180,E1 27593.001,E2 27593.001} C_VEL
LIN {X 0,Y 591.969,Z 266.559,A -85,B 0,C 180,E1 27592.325,E2 27592.325} C_VEL
LIN {X 0,Y 592.017,Z 266.486,A -85,B 0,C 180,E1 27589.168,E2 27589.168} C_VEL
LIN {X 0,Y 591.965,Z 266.493,A -85,B 0,C 180,E1 27586.155,E2 27586.155} C_VEL
LIN {X 0,Y 592.009,Z 266.489,A -85,B 0,C 180,E1 27583.006,E2 27583.006} C_VEL
LIN {X 0,Y 591.969,Z 266.492,A -85,B 0,C 180,E1 27580.055,E2 27580.055} C_VEL
LIN {X 0,Y 592,Z 266.489,A -85,B 0,C 180,E1 27576.818,E2 27576.818} C_VEL
LIN {X 0,Y 591.977,Z 266.491,A -85,B 0,C 180,E1 27573.874,E2 27573.874} C_VEL
LIN {X 0,Y 591.985,Z 266.488,A -85,B 0,C 180,E1 27570.53,E2 27570.53} C_VEL
LIN {X 0,Y 592,Z 266.492,A -85,B 0,C 180,E1 27567.542,E2 27567.542} C_VEL
LIN {X 0,Y 591.981,Z 266.489,A -85,B 0,C 180,E1 27564.338,E2 27564.338} C_VEL
LIN {X 0,Y 592.021,Z 266.492,A -85,B 0,C 180,E1 27561.291,E2 27561.291} C_VEL
LIN {X 0,Y 591.978,Z 266.489,A -85,B 0,C 180,E1 27558.106,E2 27558.106} C_VEL
LIN {X 0,Y 592.04,Z 266.488,A -85,B 0,C 180,E1 27554.975,E2 27554.975} C_VEL
LIN {X 0,Y 591.98,Z 266.49,A -85,B 0,C 180,E1 27551.793,E2 27551.793} C_VEL
LIN {X 0,Y 592.034,Z 266.485,A -85,B 0,C 180,E1 27548.645,E2 27548.645} C_VEL
LIN {X 0,Y 591.989,Z 266.491,A -85,B 0,C 180,E1 27545.525,E2 27545.525} C_VEL
LIN {X 0,Y 592.005,Z 266.485,A -85,B 0,C 180,E1 27542.226,E2 27542.226} C_VEL
LIN {X 0,Y 592.016,Z 266.492,A -85,B 0,C 180,E1 27539.129,E2 27539.129} C_VEL
LIN {X 0,Y 591.993,Z 266.485,A -85,B 0,C 180,E1 27535.932,E2 27535.932} C_VEL
LIN {X 0,Y 592.037,Z 266.491,A -85,B 0,C 180,E1 27532.821,E2 27532.821} C_VEL
LIN {X 0,Y 592.009,Z 266.483,A -85,B 0,C 180,E1 27530.054,E2 27530.054} C_VEL
LIN {X 0,Y 590.989,Z 266.613,A -85,B 0,C 180,E1 27529.308,E2 27529.308} C_VEL
LIN {X 0,Y 584.624,Z 267.419,A -85,B 0,C 180,E1 27527.216,E2 27527.216} C_VEL
LIN {X 0,Y 584.098,Z 267.478,A -85,B 0,C 180,E1 27526.672,E2 27526.672} C_VEL
LIN {X 0,Y 584.054,Z 267.475,A -85,B 0,C 180,E1 27523.466,E2 27523.466} C_VEL
LIN {X 0,Y 584.098,Z 267.475,A -85,B 0,C 180,E1 27520.292,E2 27520.292} C_VEL
LIN {X 0,Y 584.068,Z 267.48,A -85,B 0,C 180,E1 27517.068,E2 27517.068} C_VEL
LIN {X 0,Y 584.067,Z 267.475,A -85,B 0,C 180,E1 27513.68,E2 27513.68} C_VEL
LIN {X 0,Y 584.098,Z 267.479,A -85,B 0,C 180,E1 27510.462,E2 27510.462} C_VEL
LIN {X 0,Y 584.061,Z 267.478,A -85,B 0,C 180,E1 27507.251,E2 27507.251} C_VEL
LIN {X 0,Y 584.097,Z 267.474,A -85,B 0,C 180,E1 27504.045,E2 27504.045} C_VEL
LIN {X 0,Y 584.075,Z 267.48,A -85,B 0,C 180,E1 27500.826,E2 27500.826} C_VEL
LIN {X 0,Y 584.073,Z 267.475,A -85,B 0,C 180,E1 27497.454,E2 27497.454} C_VEL
LIN {X 0,Y 584.095,Z 267.48,A -85,B 0,C 180,E1 27494.299,E2 27494.299} C_VEL
LIN {X 0,Y 584.068,Z 267.477,A -85,B 0,C 180,E1 27491.098,E2 27491.098} C_VEL
LIN {X 0,Y 584.092,Z 267.475,A -85,B 0,C 180,E1 27487.894,E2 27487.894} C_VEL
LIN {X 0,Y 584.079,Z 267.48,A -85,B 0,C 180,E1 27484.633,E2 27484.633} C_VEL
LIN {X 0,Y 584.08,Z 267.473,A -85,B 0,C 180,E1 27481.243,E2 27481.243} C_VEL
LIN {X 0,Y 584.092,Z 267.479,A -85,B 0,C 180,E1 27478.082,E2 27478.082} C_VEL
LIN {X 0,Y 584.073,Z 267.476,A -85,B 0,C 180,E1 27474.867,E2 27474.867} C_VEL
LIN {X 0,Y 584.088,Z 267.474,A -85,B 0,C 180,E1 27471.64,E2 27471.64} C_VEL
LIN {X 0,Y 584.089,Z 267.48,A -85,B 0,C 180,E1 27468.359,E2 27468.359} C_VEL
LIN {X 0,Y 584.084,Z 267.474,A -85,B 0,C 180,E1 27464.98,E2 27464.98} C_VEL
LIN {X 0,Y 584.085,Z 267.478,A -85,B 0,C 180,E1 27461.754,E2 27461.754} C_VEL
LIN {X 0,Y 584.078,Z 267.477,A -85,B 0,C 180,E1 27458.565,E2 27458.565} C_VEL
LIN {X 0,Y 584.085,Z 267.474,A -85,B 0,C 180,E1 27455.402,E2 27455.402} C_VEL
LIN {X 0,Y 584.095,Z 267.481,A -85,B 0,C 180,E1 27452.06,E2 27452.06} C_VEL
LIN {X 0,Y 584.087,Z 267.473,A -85,B 0,C 180,E1 27448.725,E2 27448.725} C_VEL
LIN {X 0,Y 584.079,Z 267.477,A -85,B 0,C 180,E1 27445.484,E2 27445.484} C_VEL
LIN {X 0,Y 584.082,Z 267.477,A -85,B 0,C 180,E1 27442.327,E2 27442.327} C_VEL
LIN {X 0,Y 584.082,Z 267.474,A -85,B 0,C 180,E1 27439.147,E2 27439.147} C_VEL
LIN {X 0,Y 584.1,Z 267.481,A -85,B 0,C 180,E1 27435.831,E2 27435.831} C_VEL
LIN {X 0,Y 584.089,Z 267.474,A -85,B 0,C 180,E1 27432.466,E2 27432.466} C_VEL
LIN {X 0,Y 584.074,Z 267.477,A -85,B 0,C 180,E1 27429.247,E2 27429.247} C_VEL
LIN {X 0,Y 584.089,Z 267.478,A -85,B 0,C 180,E1 27426.066,E2 27426.066} C_VEL
LIN {X 0,Y 584.081,Z 267.473,A -85,B 0,C 180,E1 27422.803,E2 27422.803} C_VEL
LIN {X 0,Y 584.083,Z 267.479,A -85,B 0,C 180,E1 27419.435,E2 27419.435} C_VEL
LIN {X 0,Y 584.09,Z 267.475,A -85,B 0,C 180,E1 27416.198,E2 27416.198} C_VEL
LIN {X 0,Y 584.069,Z 267.477,A -85,B 0,C 180,E1 27413.069,E2 27413.069} C_VEL
LIN {X 0,Y 584.091,Z 267.477,A -85,B 0,C 180,E1 27409.923,E2 27409.923} C_VEL
LIN {X 0,Y 584.068,Z 267.476,A -85,B 0,C 180,E1 27406.785,E2 27406.785} C_VEL
LIN {X 0,Y 584.094,Z 267.482,A -85,B 0,C 180,E1 27403.483,E2 27403.483} C_VEL
LIN {X 0,Y 584.092,Z 267.473,A -85,B 0,C 180,E1 27400.192,E2 27400.192} C_VEL
LIN {X 0,Y 584.065,Z 267.478,A -85,B 0,C 180,E1 27396.924,E2 27396.924} C_VEL
LIN {X 0,Y 584.095,Z 267.478,A -85,B 0,C 180,E1 27393.685,E2 27393.685} C_VEL
LIN {X 0,Y 584.062,Z 267.476,A -85,B 0,C 180,E1 27390.56,E2 27390.56} C_VEL
LIN {X 0,Y 584.092,Z 267.482,A -85,B 0,C 180,E1 27387.307,E2 27387.307} C_VEL
LIN {X 0,Y 584.085,Z 267.474,A -85,B 0,C 180,E1 27384.043,E2 27384.043} C_VEL
LIN {X 0,Y 584.059,Z 267.479,A -85,B 0,C 180,E1 27380.755,E2 27380.755} C_VEL
LIN {X 0,Y 584.097,Z 267.477,A -85,B 0,C 180,E1 27377.534,E2 27377.534} C_VEL
LIN {X 0,Y 584.053,Z 267.475,A -85,B 0,C 180,E1 27374.373,E2 27374.373} C_VEL
LIN {X 0,Y 584.092,Z 267.479,A -85,B 0,C 180,E1 27371.153,E2 27371.153} C_VEL
LIN {X 0,Y 584.066,Z 267.474,A -85,B 0,C 180,E1 27367.97,E2 27367.97} C_VEL
LIN {X 0,Y 584.055,Z 267.476,A -85,B 0,C 180,E1 27364.615,E2 27364.615} C_VEL
LIN {X 0,Y 584.098,Z 267.473,A -85,B 0,C 180,E1 27361.471,E2 27361.471} C_VEL
LIN {X 0,Y 584.046,Z 267.476,A -85,B 0,C 180,E1 27358.332,E2 27358.332} C_VEL
LIN {X 0,Y 584.1,Z 267.476,A -85,B 0,C 180,E1 27355.189,E2 27355.189} C_VEL
LIN {X 0,Y 584.044,Z 267.475,A -85,B 0,C 180,E1 27352.029,E2 27352.029} C_VEL
LIN {X 0,Y 584.079,Z 267.482,A -85,B 0,C 180,E1 27348.773,E2 27348.773} C_VEL
LIN {X 0,Y 584.055,Z 267.474,A -85,B 0,C 180,E1 27345.678,E2 27345.678} C_VEL
LIN {X 0,Y 584.047,Z 267.48,A -85,B 0,C 180,E1 27342.361,E2 27342.361} C_VEL
LIN {X 0,Y 584.074,Z 267.473,A -85,B 0,C 180,E1 27339.351,E2 27339.351} C_VEL
LIN {X 0,Y 584.039,Z 267.48,A -85,B 0,C 180,E1 27336.17,E2 27336.17} C_VEL
LIN {X 0,Y 584.09,Z 267.474,A -85,B 0,C 180,E1 27333.105,E2 27333.105} C_VEL
LIN {X 0,Y 584.034,Z 267.477,A -85,B 0,C 180,E1 27330.007,E2 27330.007} C_VEL
LIN {X 0,Y 584.097,Z 267.479,A -85,B 0,C 180,E1 27326.903,E2 27326.903} C_VEL
LIN {X 0,Y 584.029,Z 267.48,A -85,B 0,C 180,E1 27323.739,E2 27323.739} C_VEL
LIN {X 0,Y 584.083,Z 267.476,A -85,B 0,C 180,E1 27320.536,E2 27320.536} C_VEL
LIN {X 0,Y 584.028,Z 267.479,A -85,B 0,C 180,E1 27317.549,E2 27317.549} C_VEL
LIN {X 0,Y 584.063,Z 267.483,A -85,B 0,C 180,E1 27314.31,E2 27314.31} C_VEL
LIN {X 0,Y 584.028,Z 267.475,A -85,B 0,C 180,E1 27311.362,E2 27311.362} C_VEL
LIN {X 0,Y 584.069,Z 267.622,A -85,B 0,C 180,E1 27308.137,E2 27308.137} C_VEL
LIN {X 0,Y 586.335,Z 275.274,A -85,B 0,C 180,E1 27307.055,E2 27307.055} C_VEL
LIN {X 0,Y 585.962,Z 303.569,A -85,B 0,C 180,E1 27303.915,E2 27303.915} C_VEL
LIN {X 0,Y 586.127,Z 306.361,A -85,B 0,C 180,E1 27303.673,E2 27303.673} C_VEL
LIN {X 0,Y 587.685,Z 312.359,A -85,B 0,C 180,E1 27303.483,E2 27303.483} C_VEL
LIN {X 0,Y 587.032,Z 534.955,A -85,B 0,C 180,E1 27300.381,E2 27300.381} C_VEL
LIN {X 0,Y 586.802,Z 608.481,A -85,B 0,C 180,E1 27299.345,E2 27299.345} C_VEL
LIN {X 0,Y 586.618,Z 630.625,A -85,B 0,C 180,E1 27298.846,E2 27298.846} C_VEL
LIN {X 0,Y 586.368,Z 652.289,A -85,B 0,C 180,E1 27298.167,E2 27298.167} C_VEL
LIN {X 0,Y 586.12,Z 674.092,A -85,B 0,C 180,E1 27297.281,E2 27297.281} C_VEL
LIN {X 0,Y 585.82,Z 693.737,A -85,B 0,C 180,E1 27296.289,E2 27296.289} C_VEL
LIN {X 0,Y 585.488,Z 714.166,A -85,B 0,C 180,E1 27295.056,E2 27295.056} C_VEL
LIN {X 0,Y 585.202,Z 733.36,A -85,B 0,C 180,E1 27293.682,E2 27293.682} C_VEL
LIN {X 0,Y 584.927,Z 751.107,A -85,B 0,C 180,E1 27292.195,E2 27292.195} C_VEL
LIN {X 0,Y 584.66,Z 768.225,A -85,B 0,C 180,E1 27290.522,E2 27290.522} C_VEL
LIN {X 0,Y 584.438,Z 783.734,A -85,B 0,C 180,E1 27288.761,E2 27288.761} C_VEL
LIN {X 0,Y 584.254,Z 797.738,A -85,B 0,C 180,E1 27286.913,E2 27286.913} C_VEL
LIN {X 0,Y 584.143,Z 809.735,A -85,B 0,C 180,E1 27285.08,E2 27285.08} C_VEL
LIN {X 0,Y 584.036,Z 820.86,A -85,B 0,C 180,E1 27283.06,E2 27283.06} C_VEL
LIN {X 0,Y 583.966,Z 830.481,A -85,B 0,C 180,E1 27280.956,E2 27280.956} C_VEL
LIN {X 0,Y 583.937,Z 838.24,A -85,B 0,C 180,E1 27278.865,E2 27278.865} C_VEL
LIN {X 0,Y 583.927,Z 843.91,A -85,B 0,C 180,E1 27276.884,E2 27276.884} C_VEL
LIN {X 0,Y 583.915,Z 848.472,A -85,B 0,C 180,E1 27274.714,E2 27274.714} C_VEL
LIN {X 0,Y 583.906,Z 851.328,A -85,B 0,C 180,E1 27272.552,E2 27272.552} C_VEL
LIN {X 0,Y 583.896,Z 852.395,A -85,B 0,C 180,E1 27270.491,E2 27270.491} C_VEL
LIN {X 0,Y 583.902,Z 851.886,A -85,B 0,C 180,E1 27268.234,E2 27268.234} C_VEL
LIN {X 0,Y 583.905,Z 849.866,A -85,B 0,C 180,E1 27266.171,E2 27266.171} C_VEL
LIN {X 0,Y 583.911,Z 846.199,A -85,B 0,C 180,E1 27264.103,E2 27264.103} C_VEL
LIN {X 0,Y 583.935,Z 840.67,A -85,B 0,C 180,E1 27261.929,E2 27261.929} C_VEL
LIN {X 0,Y 583.962,Z 834.046,A -85,B 0,C 180,E1 27259.942,E2 27259.942} C_VEL
LIN {X 0,Y 584.006,Z 825.224,A -85,B 0,C 180,E1 27257.844,E2 27257.844} C_VEL
LIN {X 0,Y 584.09,Z 814.983,A -85,B 0,C 180,E1 27255.831,E2 27255.831} C_VEL
LIN {X 0,Y 584.221,Z 802.685,A -85,B 0,C 180,E1 27253.802,E2 27253.802} C_VEL
LIN {X 0,Y 584.362,Z 789.462,A -85,B 0,C 180,E1 27251.96,E2 27251.96} C_VEL
LIN {X 0,Y 584.553,Z 774.665,A -85,B 0,C 180,E1 27250.178,E2 27250.178} C_VEL
LIN {X 0,Y 584.801,Z 757.967,A -85,B 0,C 180,E1 27248.45,E2 27248.45} C_VEL
LIN {X 0,Y 585.093,Z 740.758,A -85,B 0,C 180,E1 27246.91,E2 27246.91} C_VEL
LIN {X 0,Y 585.392,Z 722.039,A -85,B 0,C 180,E1 27245.478,E2 27245.478} C_VEL
LIN {X 0,Y 585.662,Z 703.094,A -85,B 0,C 180,E1 27244.248,E2 27244.248} C_VEL
LIN {X 0,Y 585.976,Z 682.395,A -85,B 0,C 180,E1 27243.118,E2 27243.118} C_VEL
LIN {X 0,Y 586.255,Z 662.551,A -85,B 0,C 180,E1 27242.224,E2 27242.224} C_VEL
LIN {X 0,Y 586.508,Z 641.344,A -85,B 0,C 180,E1 27241.467,E2 27241.467} C_VEL
LIN {X 0,Y 586.722,Z 619.105,A -85,B 0,C 180,E1 27240.87,E2 27240.87} C_VEL
LIN {X 0,Y 586.857,Z 597.65,A -85,B 0,C 180,E1 27240.479,E2 27240.479} C_VEL
LIN {X 0,Y 587.503,Z 373.192,A -85,B 0,C 180,E1 27237.375,E2 27237.375} C_VEL
LIN {X 0,Y 587.485,Z 310.933,A -85,B 0,C 180,E1 27236.484,E2 27236.484} C_VEL
LIN {X 0,Y 586.001,Z 305.679,A -85,B 0,C 180,E1 27236.292,E2 27236.292} C_VEL
LIN {X 0,Y 586.297,Z 278.202,A -85,B 0,C 180,E1 27233.276,E2 27233.276} C_VEL
LIN {X 0,Y 586.153,Z 274.181,A -85,B 0,C 180,E1 27232.807,E2 27232.807} C_VEL
LIN {X 0,Y 584.061,Z 267.544,A -85,B 0,C 180,E1 27231.831,E2 27231.831} C_VEL
LIN {X 0,Y 584.025,Z 267.475,A -85,B 0,C 180,E1 27228.578,E2 27228.578} C_VEL
LIN {X 0,Y 584.081,Z 267.483,A -85,B 0,C 180,E1 27225.548,E2 27225.548} C_VEL
LIN {X 0,Y 584.027,Z 267.479,A -85,B 0,C 180,E1 27222.418,E2 27222.418} C_VEL
LIN {X 0,Y 584.098,Z 267.471,A -85,B 0,C 180,E1 27219.299,E2 27219.299} C_VEL
LIN {X 0,Y 584.028,Z 267.48,A -85,B 0,C 180,E1 27216.202,E2 27216.202} C_VEL
LIN {X 0,Y 584.097,Z 267.479,A -85,B 0,C 180,E1 27213.097,E2 27213.097} C_VEL
LIN {X 0,Y 584.035,Z 267.477,A -85,B 0,C 180,E1 27209.975,E2 27209.975} C_VEL
LIN {X 0,Y 584.074,Z 267.474,A -85,B 0,C 180,E1 27206.758,E2 27206.758} C_VEL
LIN {X 0,Y 584.044,Z 267.48,A -85,B 0,C 180,E1 27203.723,E2 27203.723} C_VEL
LIN {X 0,Y 584.047,Z 267.474,A -85,B 0,C 180,E1 27200.336,E2 27200.336} C_VEL
LIN {X 0,Y 584.087,Z 267.481,A -85,B 0,C 180,E1 27197.22,E2 27197.22} C_VEL
LIN {X 0,Y 584.042,Z 267.475,A -85,B 0,C 180,E1 27194.069,E2 27194.069} C_VEL
LIN {X 0,Y 584.101,Z 267.477,A -85,B 0,C 180,E1 27190.953,E2 27190.953} C_VEL
LIN {X 0,Y 584.043,Z 267.476,A -85,B 0,C 180,E1 27187.773,E2 27187.773} C_VEL
LIN {X 0,Y 584.098,Z 267.473,A -85,B 0,C 180,E1 27184.615,E2 27184.615} C_VEL
LIN {X 0,Y 584.053,Z 267.476,A -85,B 0,C 180,E1 27181.471,E2 27181.471} C_VEL
LIN {X 0,Y 584.066,Z 267.474,A -85,B 0,C 180,E1 27178.136,E2 27178.136} C_VEL
LIN {X 0,Y 584.087,Z 267.478,A -85,B 0,C 180,E1 27174.992,E2 27174.992} C_VEL
LIN {X 0,Y 584.051,Z 267.476,A -85,B 0,C 180,E1 27171.732,E2 27171.732} C_VEL
LIN {X 0,Y 584.099,Z 267.477,A -85,B 0,C 180,E1 27168.547,E2 27168.547} C_VEL
LIN {X 0,Y 584.098,Z 267.478,A -85,B 0,C 180,E1 27166.672,E2 27166.672} C_VEL
LIN {X 0,Y 583.096,Z 267.598,A -85,B 0,C 180,E1 27165.916,E2 27165.916} C_VEL
LIN {X 0,Y 576.633,Z 268.399,A -85,B 0,C 180,E1 27163.796,E2 27163.796} C_VEL
LIN {X 0,Y 576.12,Z 268.464,A -85,B 0,C 180,E1 27163.244,E2 27163.244} C_VEL
LIN {X 0,Y 576.135,Z 268.464,A -85,B 0,C 180,E1 27159.902,E2 27159.902} C_VEL
LIN {X 0,Y 576.16,Z 268.47,A -85,B 0,C 180,E1 27156.634,E2 27156.634} C_VEL
LIN {X 0,Y 576.119,Z 268.467,A -85,B 0,C 180,E1 27153.35,E2 27153.35} C_VEL
LIN {X 0,Y 576.16,Z 268.463,A -85,B 0,C 180,E1 27150.129,E2 27150.129} C_VEL
LIN {X 0,Y 576.138,Z 268.469,A -85,B 0,C 180,E1 27146.862,E2 27146.862} C_VEL
LIN {X 0,Y 576.136,Z 268.464,A -85,B 0,C 180,E1 27143.593,E2 27143.593} C_VEL
LIN {X 0,Y 576.156,Z 268.468,A -85,B 0,C 180,E1 27140.311,E2 27140.311} C_VEL
LIN {X 0,Y 576.127,Z 268.467,A -85,B 0,C 180,E1 27137.084,E2 27137.084} C_VEL
LIN {X 0,Y 576.16,Z 268.462,A -85,B 0,C 180,E1 27133.787,E2 27133.787} C_VEL
LIN {X 0,Y 576.161,Z 268.47,A -85,B 0,C 180,E1 27130.374,E2 27130.374} C_VEL
LIN {X 0,Y 576.132,Z 268.465,A -85,B 0,C 180,E1 27127.152,E2 27127.152} C_VEL
LIN {X 0,Y 576.149,Z 268.466,A -85,B 0,C 180,E1 27123.95,E2 27123.95} C_VEL
LIN {X 0,Y 576.137,Z 268.468,A -85,B 0,C 180,E1 27120.678,E2 27120.678} C_VEL
LIN {X 0,Y 576.151,Z 268.461,A -85,B 0,C 180,E1 27117.311,E2 27117.311} C_VEL
LIN {X 0,Y 576.151,Z 268.467,A -85,B 0,C 180,E1 27113.958,E2 27113.958} C_VEL
LIN {X 0,Y 576.136,Z 268.466,A -85,B 0,C 180,E1 27110.734,E2 27110.734} C_VEL
LIN {X 0,Y 576.153,Z 268.463,A -85,B 0,C 180,E1 27107.471,E2 27107.471} C_VEL
LIN {X 0,Y 576.158,Z 268.47,A -85,B 0,C 180,E1 27104.061,E2 27104.061} C_VEL
LIN {X 0,Y 576.141,Z 268.464,A -85,B 0,C 180,E1 27100.802,E2 27100.802} C_VEL
LIN {X 0,Y 576.144,Z 268.465,A -85,B 0,C 180,E1 27097.579,E2 27097.579} C_VEL
LIN {X 0,Y 576.144,Z 268.467,A -85,B 0,C 180,E1 27094.379,E2 27094.379} C_VEL
LIN {X 0,Y 576.156,Z 268.46,A -85,B 0,C 180,E1 27090.994,E2 27090.994} C_VEL
LIN {X 0,Y 576.147,Z 268.468,A -85,B 0,C 180,E1 27087.713,E2 27087.713} C_VEL
LIN {X 0,Y 576.144,Z 268.466,A -85,B 0,C 180,E1 27084.423,E2 27084.423} C_VEL
LIN {X 0,Y 576.142,Z 268.464,A -85,B 0,C 180,E1 27081.216,E2 27081.216} C_VEL
LIN {X 0,Y 576.157,Z 268.47,A -85,B 0,C 180,E1 27077.879,E2 27077.879} C_VEL
LIN {X 0,Y 576.151,Z 268.463,A -85,B 0,C 180,E1 27074.5,E2 27074.5} C_VEL
LIN {X 0,Y 576.136,Z 268.466,A -85,B 0,C 180,E1 27071.274,E2 27071.274} C_VEL
LIN {X 0,Y 576.153,Z 268.468,A -85,B 0,C 180,E1 27067.986,E2 27067.986} C_VEL
LIN {X 0,Y 576.155,Z 268.461,A -85,B 0,C 180,E1 27064.619,E2 27064.619} C_VEL
LIN {X 0,Y 576.136,Z 268.467,A -85,B 0,C 180,E1 27061.268,E2 27061.268} C_VEL
LIN {X 0,Y 576.151,Z 268.466,A -85,B 0,C 180,E1 27058.043,E2 27058.043} C_VEL
LIN {X 0,Y 576.135,Z 268.464,A -85,B 0,C 180,E1 27054.819,E2 27054.819} C_VEL
LIN {X 0,Y 576.151,Z 268.47,A -85,B 0,C 180,E1 27051.465,E2 27051.465} C_VEL
LIN {X 0,Y 576.158,Z 268.462,A -85,B 0,C 180,E1 27048.212,E2 27048.212} C_VEL
LIN {X 0,Y 576.128,Z 268.466,A -85,B 0,C 180,E1 27044.923,E2 27044.923} C_VEL
LIN {X 0,Y 576.155,Z 268.469,A -85,B 0,C 180,E1 27041.656,E2 27041.656} C_VEL
LIN {X 0,Y 576.144,Z 268.463,A -85,B 0,C 180,E1 27038.335,E2 27038.335} C_VEL
LIN {X 0,Y 576.129,Z 268.468,A -85,B 0,C 180,E1 27035.003,E2 27035.003} C_VEL
LIN {X 0,Y 576.157,Z 268.465,A -85,B 0,C 180,E1 27031.754,E2 27031.754} C_VEL
LIN {X 0,Y 576.122,Z 268.466,A -85,B 0,C 180,E1 27028.581,E2 27028.581} C_VEL
LIN {X 0,Y 576.153,Z 268.471,A -85,B 0,C 180,E1 27025.271,E2 27025.271} C_VEL
LIN {X 0,Y 576.146,Z 268.463,A -85,B 0,C 180,E1 27022.015,E2 27022.015} C_VEL
LIN {X 0,Y 576.12,Z 268.468,A -85,B 0,C 180,E1 27018.727,E2 27018.727} C_VEL
LIN {X 0,Y 576.159,Z 268.462,A -85,B 0,C 180,E1 27015.501,E2 27015.501} C_VEL
LIN {X 0,Y 576.115,Z 268.466,A -85,B 0,C 180,E1 27012.294,E2 27012.294} C_VEL
LIN {X 0,Y 576.143,Z 268.467,A -85,B 0,C 180,E1 27008.986,E2 27008.986} C_VEL
LIN {X 0,Y 576.141,Z 268.464,A -85,B 0,C 180,E1 27005.777,E2 27005.777} C_VEL
LIN {X 0,Y 576.112,Z 268.466,A -85,B 0,C 180,E1 27002.487,E2 27002.487} C_VEL
LIN {X 0,Y 576.162,Z 268.466,A -85,B 0,C 180,E1 26999.304,E2 26999.304} C_VEL
LIN {X 0,Y 576.107,Z 268.464,A -85,B 0,C 180,E1 26996.119,E2 26996.119} C_VEL
LIN {X 0,Y 576.152,Z 268.468,A -85,B 0,C 180,E1 26992.922,E2 26992.922} C_VEL
LIN {X 0,Y 576.118,Z 268.463,A -85,B 0,C 180,E1 26989.739,E2 26989.739} C_VEL
LIN {X 0,Y 576.109,Z 268.465,A -85,B 0,C 180,E1 26986.379,E2 26986.379} C_VEL
LIN {X 0,Y 576.155,Z 268.463,A -85,B 0,C 180,E1 26983.257,E2 26983.257} C_VEL
LIN {X 0,Y 576.099,Z 268.464,A -85,B 0,C 180,E1 26980.113,E2 26980.113} C_VEL
LIN {X 0,Y 576.163,Z 268.468,A -85,B 0,C 180,E1 26976.909,E2 26976.909} C_VEL
LIN {X 0,Y 576.096,Z 268.464,A -85,B 0,C 180,E1 26973.801,E2 26973.801} C_VEL
LIN {X 0,Y 576.138,Z 268.467,A -85,B 0,C 180,E1 26970.585,E2 26970.585} C_VEL
LIN {X 0,Y 576.102,Z 268.469,A -85,B 0,C 180,E1 26967.507,E2 26967.507} C_VEL
LIN {X 0,Y 576.101,Z 268.47,A -85,B 0,C 180,E1 26964.143,E2 26964.143} C_VEL
LIN {X 0,Y 576.128,Z 268.456,A -85,B 0,C 180,E1 26961.08,E2 26961.08} C_VEL
LIN {X 0,Y 576.092,Z 268.469,A -85,B 0,C 180,E1 26957.938,E2 26957.938} C_VEL
LIN {X 0,Y 576.135,Z 268.463,A -85,B 0,C 180,E1 26954.922,E2 26954.922} C_VEL
LIN {X 0,Y 576.083,Z 268.46,A -85,B 0,C 180,E1 26951.728,E2 26951.728} C_VEL
LIN {X 0,Y 576.179,Z 268.66,A -85,B 0,C 180,E1 26948.624,E2 26948.624} C_VEL
LIN {X 0,Y 579.156,Z 278.119,A -85,B 0,C 180,E1 26947.262,E2 26947.262} C_VEL
LIN {X 0,Y 578.735,Z 305.58,A -85,B 0,C 180,E1 26944.196,E2 26944.196} C_VEL
LIN {X 0,Y 581,Z 314.333,A -85,B 0,C 180,E1 26943.891,E2 26943.891} C_VEL
LIN {X 0,Y 580.125,Z 535.846,A -85,B 0,C 180,E1 26940.769,E2 26940.769} C_VEL
LIN {X 0,Y 579.82,Z 608.46,A -85,B 0,C 180,E1 26939.734,E2 26939.734} C_VEL
LIN {X 0,Y 579.569,Z 631.021,A -85,B 0,C 180,E1 26939.22,E2 26939.22} C_VEL
LIN {X 0,Y 579.235,Z 652.878,A -85,B 0,C 180,E1 26938.524,E2 26938.524} C_VEL
LIN {X 0,Y 578.888,Z 674.741,A -85,B 0,C 180,E1 26937.619,E2 26937.619} C_VEL
LIN {X 0,Y 578.496,Z 693.736,A -85,B 0,C 180,E1 26936.648,E2 26936.648} C_VEL
LIN {X 0,Y 578.068,Z 714.173,A -85,B 0,C 180,E1 26935.4,E2 26935.4} C_VEL
LIN {X 0,Y 577.671,Z 733.473,A -85,B 0,C 180,E1 26934,E2 26934} C_VEL
LIN {X 0,Y 577.283,Z 751.765,A -85,B 0,C 180,E1 26932.446,E2 26932.446} C_VEL
LIN {X 0,Y 576.922,Z 768.648,A -85,B 0,C 180,E1 26930.765,E2 26930.765} C_VEL
LIN {X 0,Y 576.629,Z 783.738,A -85,B 0,C 180,E1 26929.025,E2 26929.025} C_VEL
LIN {X 0,Y 576.384,Z 798.121,A -85,B 0,C 180,E1 26927.095,E2 26927.095} C_VEL
LIN {X 0,Y 576.224,Z 810.353,A -85,B 0,C 180,E1 26925.189,E2 26925.189} C_VEL
LIN {X 0,Y 576.076,Z 821.899,A -85,B 0,C 180,E1 26923.04,E2 26923.04} C_VEL
LIN {X 0,Y 575.989,Z 830.891,A -85,B 0,C 180,E1 26921.008,E2 26921.008} C_VEL
LIN {X 0,Y 575.946,Z 838.543,A -85,B 0,C 180,E1 26918.888,E2 26918.888} C_VEL
LIN {X 0,Y 575.931,Z 844.165,A -85,B 0,C 180,E1 26916.88,E2 26916.88} C_VEL
LIN {X 0,Y 575.916,Z 848.633,A -85,B 0,C 180,E1 26914.68,E2 26914.68} C_VEL
LIN {X 0,Y 575.908,Z 851.405,A -85,B 0,C 180,E1 26912.488,E2 26912.488} C_VEL
LIN {X 0,Y 575.897,Z 852.417,A -85,B 0,C 180,E1 26910.398,E2 26910.398} C_VEL
LIN {X 0,Y 575.903,Z 851.888,A -85,B 0,C 180,E1 26908.209,E2 26908.209} C_VEL
LIN {X 0,Y 575.908,Z 849.862,A -85,B 0,C 180,E1 26906.118,E2 26906.118} C_VEL
LIN {X 0,Y 575.916,Z 846.202,A -85,B 0,C 180,E1 26904.021,E2 26904.021} C_VEL
LIN {X 0,Y 575.946,Z 840.669,A -85,B 0,C 180,E1 26901.816,E2 26901.816} C_VEL
LIN {X 0,Y 575.981,Z 834.043,A -85,B 0,C 180,E1 26899.801,E2 26899.801} C_VEL
LIN {X 0,Y 576.044,Z 825.227,A -85,B 0,C 180,E1 26897.673,E2 26897.673} C_VEL
LIN {X 0,Y 576.161,Z 814.986,A -85,B 0,C 180,E1 26895.632,E2 26895.632} C_VEL
LIN {X 0,Y 576.33,Z 802.943,A -85,B 0,C 180,E1 26893.614,E2 26893.614} C_VEL
LIN {X 0,Y 576.532,Z 789.464,A -85,B 0,C 180,E1 26891.706,E2 26891.706} C_VEL
LIN {X 0,Y 576.79,Z 774.903,A -85,B 0,C 180,E1 26889.927,E2 26889.927} C_VEL
LIN {X 0,Y 577.114,Z 758.721,A -85,B 0,C 180,E1 26888.221,E2 26888.221} C_VEL
LIN {X 0,Y 577.507,Z 741.406,A -85,B 0,C 180,E1 26886.643,E2 26886.643} C_VEL
LIN {X 0,Y 577.922,Z 722.029,A -85,B 0,C 180,E1 26885.14,E2 26885.14} C_VEL
LIN {X 0,Y 578.301,Z 703.099,A -85,B 0,C 180,E1 26883.896,E2 26883.896} C_VEL
LIN {X 0,Y 578.712,Z 682.394,A -85,B 0,C 180,E1 26882.752,E2 26882.752} C_VEL
LIN {X 0,Y 579.092,Z 662.538,A -85,B 0,C 180,E1 26881.85,E2 26881.85} C_VEL
LIN {X 0,Y 579.425,Z 641.123,A -85,B 0,C 180,E1 26881.077,E2 26881.077} C_VEL
LIN {X 0,Y 579.713,Z 618.786,A -85,B 0,C 180,E1 26880.477,E2 26880.477} C_VEL
LIN {X 0,Y 579.907,Z 596.78,A -85,B 0,C 180,E1 26880.075,E2 26880.075} C_VEL
LIN {X 0,Y 580.764,Z 372.619,A -85,B 0,C 180,E1 26876.94,E2 26876.94} C_VEL
LIN {X 0,Y 580.804,Z 312.876,A -85,B 0,C 180,E1 26876.075,E2 26876.075} C_VEL
LIN {X 0,Y 578.732,Z 305.554,A -85,B 0,C 180,E1 26875.802,E2 26875.802} C_VEL
LIN {X 0,Y 579.159,Z 277.969,A -85,B 0,C 180,E1 26872.72,E2 26872.72} C_VEL
LIN {X 0,Y 576.165,Z 268.556,A -85,B 0,C 180,E1 26871.339,E2 26871.339} C_VEL
LIN {X 0,Y 576.085,Z 268.46,A -85,B 0,C 180,E1 26868.206,E2 26868.206} C_VEL
LIN {X 0,Y 576.134,Z 268.463,A -85,B 0,C 180,E1 26865.064,E2 26865.064} C_VEL
LIN {X 0,Y 576.093,Z 268.469,A -85,B 0,C 180,E1 26862.029,E2 26862.029} C_VEL
LIN {X 0,Y 576.115,Z 268.457,A -85,B 0,C 180,E1 26858.794,E2 26858.794} C_VEL
LIN {X 0,Y 576.105,Z 268.47,A -85,B 0,C 180,E1 26855.794,E2 26855.794} C_VEL
LIN {X 0,Y 576.099,Z 268.469,A -85,B 0,C 180,E1 26852.431,E2 26852.431} C_VEL
LIN {X 0,Y 576.153,Z 268.467,A -85,B 0,C 180,E1 26849.3,E2 26849.3} C_VEL
LIN {X 0,Y 576.095,Z 268.464,A -85,B 0,C 180,E1 26846.157,E2 26846.157} C_VEL
LIN {X 0,Y 576.164,Z 268.466,A -85,B 0,C 180,E1 26842.983,E2 26842.983} C_VEL
LIN {X 0,Y 576.1,Z 268.463,A -85,B 0,C 180,E1 26839.839,E2 26839.839} C_VEL
LIN {X 0,Y 576.144,Z 268.463,A -85,B 0,C 180,E1 26836.639,E2 26836.639} C_VEL
LIN {X 0,Y 576.112,Z 268.465,A -85,B 0,C 180,E1 26833.55,E2 26833.55} C_VEL
LIN {X 0,Y 576.113,Z 268.463,A -85,B 0,C 180,E1 26830.196,E2 26830.196} C_VEL
LIN {X 0,Y 576.152,Z 268.468,A -85,B 0,C 180,E1 26827.078,E2 26827.078} C_VEL
LIN {X 0,Y 576.107,Z 268.464,A -85,B 0,C 180,E1 26823.881,E2 26823.881} C_VEL
LIN {X 0,Y 576.162,Z 268.466,A -85,B 0,C 180,E1 26820.696,E2 26820.696} C_VEL
LIN {X 0,Y 576.112,Z 268.466,A -85,B 0,C 180,E1 26817.513,E2 26817.513} C_VEL
LIN {X 0,Y 576.141,Z 268.464,A -85,B 0,C 180,E1 26814.223,E2 26814.223} C_VEL
LIN {X 0,Y 576.143,Z 268.467,A -85,B 0,C 180,E1 26811.014,E2 26811.014} C_VEL
LIN {X 0,Y 576.115,Z 268.466,A -85,B 0,C 180,E1 26807.706,E2 26807.706} C_VEL
LIN {X 0,Y 576.159,Z 268.462,A -85,B 0,C 180,E1 26804.499,E2 26804.499} C_VEL
LIN {X 0,Y 576.12,Z 268.464,A -85,B 0,C 180,E1 26803.244,E2 26803.244} C_VEL
LIN {X 0,Y 575.167,Z 268.59,A -85,B 0,C 180,E1 26802.478,E2 26802.478} C_VEL
LIN {X 0,Y 568.646,Z 269.401,A -85,B 0,C 180,E1 26800.272,E2 26800.272} C_VEL
LIN {X 0,Y 568.188,Z 269.453,A -85,B 0,C 180,E1 26799.767,E2 26799.767} C_VEL
LIN {X 0,Y 568.222,Z 269.458,A -85,B 0,C 180,E1 26796.567,E2 26796.567} C_VEL
LIN {X 0,Y 568.182,Z 269.456,A -85,B 0,C 180,E1 26793.337,E2 26793.337} C_VEL
LIN {X 0,Y 568.225,Z 269.451,A -85,B 0,C 180,E1 26790.018,E2 26790.018} C_VEL
LIN {X 0,Y 568.213,Z 269.46,A -85,B 0,C 180,E1 26786.701,E2 26786.701} C_VEL
LIN {X 0,Y 568.187,Z 269.455,A -85,B 0,C 180,E1 26783.361,E2 26783.361} C_VEL
LIN {X 0,Y 568.217,Z 269.454,A -85,B 0,C 180,E1 26780.101,E2 26780.101} C_VEL
LIN {X 0,Y 568.198,Z 269.458,A -85,B 0,C 180,E1 26776.802,E2 26776.802} C_VEL
LIN {X 0,Y 568.198,Z 269.453,A -85,B 0,C 180,E1 26773.385,E2 26773.385} C_VEL
LIN {X 0,Y 568.214,Z 269.456,A -85,B 0,C 180,E1 26770.092,E2 26770.092} C_VEL
LIN {X 0,Y 568.193,Z 269.456,A -85,B 0,C 180,E1 26766.873,E2 26766.873} C_VEL
LIN {X 0,Y 568.217,Z 269.45,A -85,B 0,C 180,E1 26763.481,E2 26763.481} C_VEL
LIN {X 0,Y 568.216,Z 269.456,A -85,B 0,C 180,E1 26760.098,E2 26760.098} C_VEL
LIN {X 0,Y 568.196,Z 269.454,A -85,B 0,C 180,E1 26756.853,E2 26756.853} C_VEL
LIN {X 0,Y 568.216,Z 269.451,A -85,B 0,C 180,E1 26753.541,E2 26753.541} C_VEL
LIN {X 0,Y 568.219,Z 269.458,A -85,B 0,C 180,E1 26750.174,E2 26750.174} C_VEL
LIN {X 0,Y 568.2,Z 269.454,A -85,B 0,C 180,E1 26746.81,E2 26746.81} C_VEL
LIN {X 0,Y 568.209,Z 269.453,A -85,B 0,C 180,E1 26743.534,E2 26743.534} C_VEL
LIN {X 0,Y 568.213,Z 269.459,A -85,B 0,C 180,E1 26740.237,E2 26740.237} C_VEL
LIN {X 0,Y 568.208,Z 269.452,A -85,B 0,C 180,E1 26736.872,E2 26736.872} C_VEL
LIN {X 0,Y 568.205,Z 269.455,A -85,B 0,C 180,E1 26733.632,E2 26733.632} C_VEL
LIN {X 0,Y 568.204,Z 269.455,A -85,B 0,C 180,E1 26730.403,E2 26730.403} C_VEL
LIN {X 0,Y 568.214,Z 269.45,A -85,B 0,C 180,E1 26727.075,E2 26727.075} C_VEL
LIN {X 0,Y 568.21,Z 269.458,A -85,B 0,C 180,E1 26723.737,E2 26723.737} C_VEL
LIN {X 0,Y 568.208,Z 269.454,A -85,B 0,C 180,E1 26720.479,E2 26720.479} C_VEL
LIN {X 0,Y 568.202,Z 269.454,A -85,B 0,C 180,E1 26717.19,E2 26717.19} C_VEL
LIN {X 0,Y 568.219,Z 269.458,A -85,B 0,C 180,E1 26713.858,E2 26713.858} C_VEL
LIN {X 0,Y 568.214,Z 269.452,A -85,B 0,C 180,E1 26710.469,E2 26710.469} C_VEL
LIN {X 0,Y 568.196,Z 269.455,A -85,B 0,C 180,E1 26707.224,E2 26707.224} C_VEL
LIN {X 0,Y 568.215,Z 269.457,A -85,B 0,C 180,E1 26703.903,E2 26703.903} C_VEL
LIN {X 0,Y 568.214,Z 269.45,A -85,B 0,C 180,E1 26700.578,E2 26700.578} C_VEL
LIN {X 0,Y 568.197,Z 269.456,A -85,B 0,C 180,E1 26697.26,E2 26697.26} C_VEL
LIN {X 0,Y 568.212,Z 269.455,A -85,B 0,C 180,E1 26694.005,E2 26694.005} C_VEL
LIN {X 0,Y 568.196,Z 269.453,A -85,B 0,C 180,E1 26690.739,E2 26690.739} C_VEL
LIN {X 0,Y 568.207,Z 269.459,A -85,B 0,C 180,E1 26687.353,E2 26687.353} C_VEL
LIN {X 0,Y 568.218,Z 269.453,A -85,B 0,C 180,E1 26684.032,E2 26684.032} C_VEL
LIN {X 0,Y 568.189,Z 269.455,A -85,B 0,C 180,E1 26680.757,E2 26680.757} C_VEL
LIN {X 0,Y 568.219,Z 269.459,A -85,B 0,C 180,E1 26677.479,E2 26677.479} C_VEL
LIN {X 0,Y 568.215,Z 269.451,A -85,B 0,C 180,E1 26674.148,E2 26674.148} C_VEL
LIN {X 0,Y 568.183,Z 269.456,A -85,B 0,C 180,E1 26670.803,E2 26670.803} C_VEL
LIN {X 0,Y 568.221,Z 269.457,A -85,B 0,C 180,E1 26667.523,E2 26667.523} C_VEL
LIN {X 0,Y 568.195,Z 269.453,A -85,B 0,C 180,E1 26664.206,E2 26664.206} C_VEL
LIN {X 0,Y 568.185,Z 269.457,A -85,B 0,C 180,E1 26660.822,E2 26660.822} C_VEL
LIN {X 0,Y 568.22,Z 269.454,A -85,B 0,C 180,E1 26657.617,E2 26657.617} C_VEL
LIN {X 0,Y 568.177,Z 269.453,A -85,B 0,C 180,E1 26654.367,E2 26654.367} C_VEL
LIN {X 0,Y 568.207,Z 269.454,A -85,B 0,C 180,E1 26651.058,E2 26651.058} C_VEL
LIN {X 0,Y 568.205,Z 269.45,A -85,B 0,C 180,E1 26647.787,E2 26647.787} C_VEL
LIN {X 0,Y 568.175,Z 269.452,A -85,B 0,C 180,E1 26644.542,E2 26644.542} C_VEL
LIN {X 0,Y 568.221,Z 269.453,A -85,B 0,C 180,E1 26641.311,E2 26641.311} C_VEL
LIN {X 0,Y 568.168,Z 269.451,A -85,B 0,C 180,E1 26638.185,E2 26638.185} C_VEL
LIN {X 0,Y 568.214,Z 269.459,A -85,B 0,C 180,E1 26634.952,E2 26634.952} C_VEL
LIN {X 0,Y 568.176,Z 269.451,A -85,B 0,C 180,E1 26631.805,E2 26631.805} C_VEL
LIN {X 0,Y 568.172,Z 269.458,A -85,B 0,C 180,E1 26628.427,E2 26628.427} C_VEL
LIN {X 0,Y 568.218,Z 269.451,A -85,B 0,C 180,E1 26625.218,E2 26625.218} C_VEL
LIN {X 0,Y 568.161,Z 269.457,A -85,B 0,C 180,E1 26622.063,E2 26622.063} C_VEL
LIN {X 0,Y 568.217,Z 269.452,A -85,B 0,C 180,E1 26618.841,E2 26618.841} C_VEL
LIN {X 0,Y 568.165,Z 269.456,A -85,B 0,C 180,E1 26615.683,E2 26615.683} C_VEL
LIN {X 0,Y 568.169,Z 269.459,A -85,B 0,C 180,E1 26612.27,E2 26612.27} C_VEL
LIN {X 0,Y 568.196,Z 269.452,A -85,B 0,C 180,E1 26609.172,E2 26609.172} C_VEL
LIN {X 0,Y 568.155,Z 269.457,A -85,B 0,C 180,E1 26605.97,E2 26605.97} C_VEL
LIN {X 0,Y 568.22,Z 269.452,A -85,B 0,C 180,E1 26602.853,E2 26602.853} C_VEL
LIN {X 0,Y 568.15,Z 269.458,A -85,B 0,C 180,E1 26599.77,E2 26599.77} C_VEL
LIN {X 0,Y 568.215,Z 269.445,A -85,B 0,C 180,E1 26596.612,E2 26596.612} C_VEL
LIN {X 0,Y 568.149,Z 269.461,A -85,B 0,C 180,E1 26593.479,E2 26593.479} C_VEL
LIN {X 0,Y 568.177,Z 269.464,A -85,B 0,C 180,E1 26590.205,E2 26590.205} C_VEL
LIN {X 0,Y 568.193,Z 269.678,A -85,B 0,C 180,E1 26589.145,E2 26589.145} C_VEL
LIN {X 0,Y 571.969,Z 281.574,A -85,B 0,C 180,E1 26587.405,E2 26587.405} C_VEL
LIN {X 0,Y 571.543,Z 305.918,A -85,B 0,C 180,E1 26584.669,E2 26584.669} C_VEL
LIN {X 0,Y 574.347,Z 316.185,A -85,B 0,C 180,E1 26584.311,E2 26584.311} C_VEL
LIN {X 0,Y 573.243,Z 536.991,A -85,B 0,C 180,E1 26581.163,E2 26581.163} C_VEL
LIN {X 0,Y 572.865,Z 608.439,A -85,B 0,C 180,E1 26580.132,E2 26580.132} C_VEL
LIN {X 0,Y 572.547,Z 631.28,A -85,B 0,C 180,E1 26579.607,E2 26579.607} C_VEL
LIN {X 0,Y 572.127,Z 653.448,A -85,B 0,C 180,E1 26578.89,E2 26578.89} C_VEL
LIN {X 0,Y 571.674,Z 675.4,A -85,B 0,C 180,E1 26577.964,E2 26577.964} C_VEL
LIN {X 0,Y 571.193,Z 693.966,A -85,B 0,C 180,E1 26577.002,E2 26577.002} C_VEL
LIN {X 0,Y 570.676,Z 714.18,A -85,B 0,C 180,E1 26575.753,E2 26575.753} C_VEL
LIN {X 0,Y 570.177,Z 732.782,A -85,B 0,C 180,E1 26574.391,E2 26574.391} C_VEL
LIN {X 0,Y 569.683,Z 750.648,A -85,B 0,C 180,E1 26572.864,E2 26572.864} C_VEL
LIN {X 0,Y 569.221,Z 767.927,A -85,B 0,C 180,E1 26571.137,E2 26571.137} C_VEL
LIN {X 0,Y 568.836,Z 783.742,A -85,B 0,C 180,E1 26569.296,E2 26569.296} C_VEL
LIN {X 0,Y 568.541,Z 797.736,A -85,B 0,C 180,E1 26567.395,E2 26567.395} C_VEL
LIN {X 0,Y 568.325,Z 809.728,A -85,B 0,C 180,E1 26565.51,E2 26565.51} C_VEL
LIN {X 0,Y 568.143,Z 820.867,A -85,B 0,C 180,E1 26563.432,E2 26563.432} C_VEL
LIN {X 0,Y 568.028,Z 830.487,A -85,B 0,C 180,E1 26561.267,E2 26561.267} C_VEL
LIN {X 0,Y 567.971,Z 838.237,A -85,B 0,C 180,E1 26559.116,E2 26559.116} C_VEL
LIN {X 0,Y 567.936,Z 843.911,A -85,B 0,C 180,E1 26557.079,E2 26557.079} C_VEL
LIN {X 0,Y 567.917,Z 848.539,A -85,B 0,C 180,E1 26554.808,E2 26554.808} C_VEL
LIN {X 0,Y 567.906,Z 851.32,A -85,B 0,C 180,E1 26552.624,E2 26552.624} C_VEL
LIN {X 0,Y 567.896,Z 852.395,A -85,B 0,C 180,E1 26550.504,E2 26550.504} C_VEL
LIN {X 0,Y 567.904,Z 851.89,A -85,B 0,C 180,E1 26548.184,E2 26548.184} C_VEL
LIN {X 0,Y 567.91,Z 849.858,A -85,B 0,C 180,E1 26546.063,E2 26546.063} C_VEL
LIN {X 0,Y 567.92,Z 846.204,A -85,B 0,C 180,E1 26543.936,E2 26543.936} C_VEL
LIN {X 0,Y 567.945,Z 840.668,A -85,B 0,C 180,E1 26541.7,E2 26541.7} C_VEL
LIN {X 0,Y 567.997,Z 834.04,A -85,B 0,C 180,E1 26539.657,E2 26539.657} C_VEL
LIN {X 0,Y 568.081,Z 825.231,A -85,B 0,C 180,E1 26537.498,E2 26537.498} C_VEL
LIN {X 0,Y 568.226,Z 814.935,A -85,B 0,C 180,E1 26535.417,E2 26535.417} C_VEL
LIN {X 0,Y 568.45,Z 802.684,A -85,B 0,C 180,E1 26533.34,E2 26533.34} C_VEL
LIN {X 0,Y 568.712,Z 789.466,A -85,B 0,C 180,E1 26531.445,E2 26531.445} C_VEL
LIN {X 0,Y 569.049,Z 774.907,A -85,B 0,C 180,E1 26529.642,E2 26529.642} C_VEL
LIN {X 0,Y 569.472,Z 758.173,A -85,B 0,C 180,E1 26527.86,E2 26527.86} C_VEL
LIN {X 0,Y 569.944,Z 741.382,A -85,B 0,C 180,E1 26526.312,E2 26526.312} C_VEL
LIN {X 0,Y 570.474,Z 722.019,A -85,B 0,C 180,E1 26524.793,E2 26524.793} C_VEL
LIN {X 0,Y 570.968,Z 703.104,A -85,B 0,C 180,E1 26523.534,E2 26523.534} C_VEL
LIN {X 0,Y 571.474,Z 682.393,A -85,B 0,C 180,E1 26522.378,E2 26522.378} C_VEL
LIN {X 0,Y 571.956,Z 662.525,A -85,B 0,C 180,E1 26521.467,E2 26521.467} C_VEL
LIN {X 0,Y 572.375,Z 640.892,A -85,B 0,C 180,E1 26520.678,E2 26520.678} C_VEL
LIN {X 0,Y 572.727,Z 618.912,A -85,B 0,C 180,E1 26520.084,E2 26520.084} C_VEL
LIN {X 0,Y 572.971,Z 596.895,A -85,B 0,C 180,E1 26519.677,E2 26519.677} C_VEL
LIN {X 0,Y 574.055,Z 372.929,A -85,B 0,C 180,E1 26516.507,E2 26516.507} C_VEL
LIN {X 0,Y 574.181,Z 314.925,A -85,B 0,C 180,E1 26515.659,E2 26515.659} C_VEL
LIN {X 0,Y 571.498,Z 305.628,A -85,B 0,C 180,E1 26515.314,E2 26515.314} C_VEL
LIN {X 0,Y 571.95,Z 281.025,A -85,B 0,C 180,E1 26512.529,E2 26512.529} C_VEL
LIN {X 0,Y 568.176,Z 269.584,A -85,B 0,C 180,E1 26510.821,E2 26510.821} C_VEL
LIN {X 0,Y 568.164,Z 269.445,A -85,B 0,C 180,E1 26507.897,E2 26507.897} C_VEL
LIN {X 0,Y 568.154,Z 269.451,A -85,B 0,C 180,E1 26504.602,E2 26504.602} C_VEL
LIN {X 0,Y 568.211,Z 269.459,A -85,B 0,C 180,E1 26501.445,E2 26501.445} C_VEL
LIN {X 0,Y 568.15,Z 269.445,A -85,B 0,C 180,E1 26498.277,E2 26498.277} C_VEL
LIN {X 0,Y 568.215,Z 269.456,A -85,B 0,C 180,E1 26495.094,E2 26495.094} C_VEL
LIN {X 0,Y 568.157,Z 269.459,A -85,B 0,C 180,E1 26491.982,E2 26491.982} C_VEL
LIN {X 0,Y 568.187,Z 269.457,A -85,B 0,C 180,E1 26488.712,E2 26488.712} C_VEL
LIN {X 0,Y 568.174,Z 269.454,A -85,B 0,C 180,E1 26485.652,E2 26485.652} C_VEL
LIN {X 0,Y 568.167,Z 269.455,A -85,B 0,C 180,E1 26482.341,E2 26482.341} C_VEL
LIN {X 0,Y 568.212,Z 269.454,A -85,B 0,C 180,E1 26479.211,E2 26479.211} C_VEL
LIN {X 0,Y 568.163,Z 269.453,A -85,B 0,C 180,E1 26476.039,E2 26476.039} C_VEL
LIN {X 0,Y 568.223,Z 269.455,A -85,B 0,C 180,E1 26472.81,E2 26472.81} C_VEL
LIN {X 0,Y 568.169,Z 269.454,A -85,B 0,C 180,E1 26469.624,E2 26469.624} C_VEL
LIN {X 0,Y 568.185,Z 269.455,A -85,B 0,C 180,E1 26466.264,E2 26466.264} C_VEL
LIN {X 0,Y 568.213,Z 269.451,A -85,B 0,C 180,E1 26463.026,E2 26463.026} C_VEL
LIN {X 0,Y 568.17,Z 269.456,A -85,B 0,C 180,E1 26459.798,E2 26459.798} C_VEL
LIN {X 0,Y 568.22,Z 269.449,A -85,B 0,C 180,E1 26456.57,E2 26456.57} C_VEL
LIN {X 0,Y 568.18,Z 269.458,A -85,B 0,C 180,E1 26453.33,E2 26453.33} C_VEL
LIN {X 0,Y 568.187,Z 269.448,A -85,B 0,C 180,E1 26449.967,E2 26449.967} C_VEL
LIN {X 0,Y 568.22,Z 269.457,A -85,B 0,C 180,E1 26446.776,E2 26446.776} C_VEL
LIN {X 0,Y 568.177,Z 269.451,A -85,B 0,C 180,E1 26443.541,E2 26443.541} C_VEL
LIN {X 0,Y 568.219,Z 269.452,A -85,B 0,C 180,E1 26440.254,E2 26440.254} C_VEL
LIN {X 0,Y 568.188,Z 269.453,A -85,B 0,C 180,E1 26439.767,E2 26439.767} C_VEL
LIN {X 0,Y 567.18,Z 269.586,A -85,B 0,C 180,E1 26438.99,E2 26438.99} C_VEL
LIN {X 0,Y 560.803,Z 270.384,A -85,B 0,C 180,E1 26436.81,E2 26436.81} C_VEL
LIN {X 0,Y 560.281,Z 270.442,A -85,B 0,C 180,E1 26436.242,E2 26436.242} C_VEL
LIN {X 0,Y 560.26,Z 270.447,A -85,B 0,C 180,E1 26432.93,E2 26432.93} C_VEL
LIN {X 0,Y 560.25,Z 270.443,A -85,B 0,C 180,E1 26429.538,E2 26429.538} C_VEL
LIN {X 0,Y 560.279,Z 270.444,A -85,B 0,C 180,E1 26426.262,E2 26426.262} C_VEL
LIN {X 0,Y 560.25,Z 270.446,A -85,B 0,C 180,E1 26423.028,E2 26423.028} C_VEL
LIN {X 0,Y 560.267,Z 270.441,A -85,B 0,C 180,E1 26419.623,E2 26419.623} C_VEL
LIN {X 0,Y 560.279,Z 270.446,A -85,B 0,C 180,E1 26416.28,E2 26416.28} C_VEL
LIN {X 0,Y 560.252,Z 270.445,A -85,B 0,C 180,E1 26412.97,E2 26412.97} C_VEL
LIN {X 0,Y 560.279,Z 270.44,A -85,B 0,C 180,E1 26409.707,E2 26409.707} C_VEL
LIN {X 0,Y 560.28,Z 270.448,A -85,B 0,C 180,E1 26406.332,E2 26406.332} C_VEL
LIN {X 0,Y 560.255,Z 270.444,A -85,B 0,C 180,E1 26402.977,E2 26402.977} C_VEL
LIN {X 0,Y 560.28,Z 270.439,A -85,B 0,C 180,E1 26399.624,E2 26399.624} C_VEL
LIN {X 0,Y 560.28,Z 270.448,A -85,B 0,C 180,E1 26396.267,E2 26396.267} C_VEL
LIN {X 0,Y 560.258,Z 270.443,A -85,B 0,C 180,E1 26392.895,E2 26392.895} C_VEL
LIN {X 0,Y 560.273,Z 270.442,A -85,B 0,C 180,E1 26389.603,E2 26389.603} C_VEL
LIN {X 0,Y 560.277,Z 270.448,A -85,B 0,C 180,E1 26386.24,E2 26386.24} C_VEL
LIN {X 0,Y 560.266,Z 270.442,A -85,B 0,C 180,E1 26382.889,E2 26382.889} C_VEL
LIN {X 0,Y 560.269,Z 270.443,A -85,B 0,C 180,E1 26379.553,E2 26379.553} C_VEL
LIN {X 0,Y 560.273,Z 270.447,A -85,B 0,C 180,E1 26376.249,E2 26376.249} C_VEL
LIN {X 0,Y 560.272,Z 270.44,A -85,B 0,C 180,E1 26372.864,E2 26372.864} C_VEL
LIN {X 0,Y 560.266,Z 270.444,A -85,B 0,C 180,E1 26369.591,E2 26369.591} C_VEL
LIN {X 0,Y 560.268,Z 270.445,A -85,B 0,C 180,E1 26366.317,E2 26366.317} C_VEL
LIN {X 0,Y 560.283,Z 270.439,A -85,B 0,C 180,E1 26362.927,E2 26362.927} C_VEL
LIN {X 0,Y 560.264,Z 270.446,A -85,B 0,C 180,E1 26359.512,E2 26359.512} C_VEL
LIN {X 0,Y 560.271,Z 270.446,A -85,B 0,C 180,E1 26356.165,E2 26356.165} C_VEL
LIN {X 0,Y 560.272,Z 270.441,A -85,B 0,C 180,E1 26352.875,E2 26352.875} C_VEL
LIN {X 0,Y 560.266,Z 270.447,A -85,B 0,C 180,E1 26349.527,E2 26349.527} C_VEL
LIN {X 0,Y 560.273,Z 270.443,A -85,B 0,C 180,E1 26346.215,E2 26346.215} C_VEL
LIN {X 0,Y 560.26,Z 270.441,A -85,B 0,C 180,E1 26342.931,E2 26342.931} C_VEL
LIN {X 0,Y 560.273,Z 270.447,A -85,B 0,C 180,E1 26339.537,E2 26339.537} C_VEL
LIN {X 0,Y 560.273,Z 270.442,A -85,B 0,C 180,E1 26336.167,E2 26336.167} C_VEL
LIN {X 0,Y 560.254,Z 270.443,A -85,B 0,C 180,E1 26332.901,E2 26332.901} C_VEL
LIN {X 0,Y 560.283,Z 270.447,A -85,B 0,C 180,E1 26329.626,E2 26329.626} C_VEL
LIN {X 0,Y 560.282,Z 270.441,A -85,B 0,C 180,E1 26326.18,E2 26326.18} C_VEL
LIN {X 0,Y 560.249,Z 270.444,A -85,B 0,C 180,E1 26322.84,E2 26322.84} C_VEL
LIN {X 0,Y 560.283,Z 270.447,A -85,B 0,C 180,E1 26319.564,E2 26319.564} C_VEL
LIN {X 0,Y 560.273,Z 270.441,A -85,B 0,C 180,E1 26316.207,E2 26316.207} C_VEL
LIN {X 0,Y 560.247,Z 270.446,A -85,B 0,C 180,E1 26312.857,E2 26312.857} C_VEL
LIN {X 0,Y 560.28,Z 270.445,A -85,B 0,C 180,E1 26309.625,E2 26309.625} C_VEL
LIN {X 0,Y 560.249,Z 270.443,A -85,B 0,C 180,E1 26306.379,E2 26306.379} C_VEL
LIN {X 0,Y 560.253,Z 270.447,A -85,B 0,C 180,E1 26302.949,E2 26302.949} C_VEL
LIN {X 0,Y 560.283,Z 270.442,A -85,B 0,C 180,E1 26299.711,E2 26299.711} C_VEL
LIN {X 0,Y 560.237,Z 270.439,A -85,B 0,C 180,E1 26296.485,E2 26296.485} C_VEL
LIN {X 0,Y 560.28,Z 270.447,A -85,B 0,C 180,E1 26293.204,E2 26293.204} C_VEL
LIN {X 0,Y 560.257,Z 270.436,A -85,B 0,C 180,E1 26289.905,E2 26289.905} C_VEL
LIN {X 0,Y 560.237,Z 270.446,A -85,B 0,C 180,E1 26286.559,E2 26286.559} C_VEL
LIN {X 0,Y 560.281,Z 270.437,A -85,B 0,C 180,E1 26283.274,E2 26283.274} C_VEL
LIN {X 0,Y 560.234,Z 270.444,A -85,B 0,C 180,E1 26280.102,E2 26280.102} C_VEL
LIN {X 0,Y 560.25,Z 270.443,A -85,B 0,C 180,E1 26276.726,E2 26276.726} C_VEL
LIN {X 0,Y 560.264,Z 270.443,A -85,B 0,C 180,E1 26273.545,E2 26273.545} C_VEL
LIN {X 0,Y 560.227,Z 270.442,A -85,B 0,C 180,E1 26270.238,E2 26270.238} C_VEL
LIN {X 0,Y 560.281,Z 270.446,A -85,B 0,C 180,E1 26266.994,E2 26266.994} C_VEL
LIN {X 0,Y 560.23,Z 270.442,A -85,B 0,C 180,E1 26263.772,E2 26263.772} C_VEL
LIN {X 0,Y 560.235,Z 270.441,A -85,B 0,C 180,E1 26260.396,E2 26260.396} C_VEL
LIN {X 0,Y 560.268,Z 270.443,A -85,B 0,C 180,E1 26257.216,E2 26257.216} C_VEL
LIN {X 0,Y 560.218,Z 270.441,A -85,B 0,C 180,E1 26253.957,E2 26253.957} C_VEL
LIN {X 0,Y 560.278,Z 270.444,A -85,B 0,C 180,E1 26250.727,E2 26250.727} C_VEL
LIN {X 0,Y 560.221,Z 270.447,A -85,B 0,C 180,E1 26247.583,E2 26247.583} C_VEL
LIN {X 0,Y 560.226,Z 270.448,A -85,B 0,C 180,E1 26244.169,E2 26244.169} C_VEL
LIN {X 0,Y 560.249,Z 270.429,A -85,B 0,C 180,E1 26241.083,E2 26241.083} C_VEL
LIN {X 0,Y 560.212,Z 270.447,A -85,B 0,C 180,E1 26237.85,E2 26237.85} C_VEL
LIN {X 0,Y 560.28,Z 270.44,A -85,B 0,C 180,E1 26234.676,E2 26234.676} C_VEL
LIN {X 0,Y 560.206,Z 270.433,A -85,B 0,C 180,E1 26231.464,E2 26231.464} C_VEL
LIN {X 0,Y 560.244,Z 270.72,A -85,B 0,C 180,E1 26229.672,E2 26229.672} C_VEL
LIN {X 0,Y 564.775,Z 284.256,A -85,B 0,C 180,E1 26227.644,E2 26227.644} C_VEL
LIN {X 0,Y 564.323,Z 305.917,A -85,B 0,C 180,E1 26225.177,E2 26225.177} C_VEL
LIN {X 0,Y 567.723,Z 318.178,A -85,B 0,C 180,E1 26224.738,E2 26224.738} C_VEL
LIN {X 0,Y 566.39,Z 538.263,A -85,B 0,C 180,E1 26221.564,E2 26221.564} C_VEL
LIN {X 0,Y 565.939,Z 608.417,A -85,B 0,C 180,E1 26220.54,E2 26220.54} C_VEL
LIN {X 0,Y 565.549,Z 631.642,A -85,B 0,C 180,E1 26220.001,E2 26220.001} C_VEL
LIN {X 0,Y 565.068,Z 653.331,A -85,B 0,C 180,E1 26219.29,E2 26219.29} C_VEL
LIN {X 0,Y 564.537,Z 674.521,A -85,B 0,C 180,E1 26218.394,E2 26218.394} C_VEL
LIN {X 0,Y 563.932,Z 693.727,A -85,B 0,C 180,E1 26217.392,E2 26217.392} C_VEL
LIN {X 0,Y 563.306,Z 714.187,A -85,B 0,C 180,E1 26216.116,E2 26216.116} C_VEL
LIN {X 0,Y 562.694,Z 732.375,A -85,B 0,C 180,E1 26214.77,E2 26214.77} C_VEL
LIN {X 0,Y 562.11,Z 749.902,A -85,B 0,C 180,E1 26213.258,E2 26213.258} C_VEL
LIN {X 0,Y 561.559,Z 767.221,A -85,B 0,C 180,E1 26211.517,E2 26211.517} C_VEL
LIN {X 0,Y 561.084,Z 782.895,A -85,B 0,C 180,E1 26209.681,E2 26209.681} C_VEL
LIN {X 0,Y 560.711,Z 797.025,A -85,B 0,C 180,E1 26207.753,E2 26207.753} C_VEL
LIN {X 0,Y 560.421,Z 809.093,A -85,B 0,C 180,E1 26205.841,E2 26205.841} C_VEL
LIN {X 0,Y 560.199,Z 820.351,A -85,B 0,C 180,E1 26203.732,E2 26203.732} C_VEL
LIN {X 0,Y 560.058,Z 830.082,A -85,B 0,C 180,E1 26201.534,E2 26201.534} C_VEL
LIN {X 0,Y 559.981,Z 837.932,A -85,B 0,C 180,E1 26199.351,E2 26199.351} C_VEL
LIN {X 0,Y 559.938,Z 843.912,A -85,B 0,C 180,E1 26197.18,E2 26197.18} C_VEL
LIN {X 0,Y 559.919,Z 848.481,A -85,B 0,C 180,E1 26194.917,E2 26194.917} C_VEL
LIN {X 0,Y 559.907,Z 851.316,A -85,B 0,C 180,E1 26192.661,E2 26192.661} C_VEL
LIN {X 0,Y 559.897,Z 852.395,A -85,B 0,C 180,E1 26190.512,E2 26190.512} C_VEL
LIN {X 0,Y 559.905,Z 851.892,A -85,B 0,C 180,E1 26188.158,E2 26188.158} C_VEL
LIN {X 0,Y 559.911,Z 849.854,A -85,B 0,C 180,E1 26186.007,E2 26186.007} C_VEL
LIN {X 0,Y 559.922,Z 846.206,A -85,B 0,C 180,E1 26183.85,E2 26183.85} C_VEL
LIN {X 0,Y 559.946,Z 840.666,A -85,B 0,C 180,E1 26181.581,E2 26181.581} C_VEL
LIN {X 0,Y 560.012,Z 834.4,A -85,B 0,C 180,E1 26179.611,E2 26179.611} C_VEL
LIN {X 0,Y 560.116,Z 825.697,A -85,B 0,C 180,E1 26177.422,E2 26177.422} C_VEL
LIN {X 0,Y 560.292,Z 815.369,A -85,B 0,C 180,E1 26175.288,E2 26175.288} C_VEL
LIN {X 0,Y 560.543,Z 803.964,A -85,B 0,C 180,E1 26173.308,E2 26173.308} C_VEL
LIN {X 0,Y 560.858,Z 791.021,A -85,B 0,C 180,E1 26171.392,E2 26171.392} C_VEL
LIN {X 0,Y 561.267,Z 776.717,A -85,B 0,C 180,E1 26169.559,E2 26169.559} C_VEL
LIN {X 0,Y 561.781,Z 759.982,A -85,B 0,C 180,E1 26167.723,E2 26167.723} C_VEL
LIN {X 0,Y 562.314,Z 743.842,A -85,B 0,C 180,E1 26166.195,E2 26166.195} C_VEL
LIN {X 0,Y 562.949,Z 724.981,A -85,B 0,C 180,E1 26164.657,E2 26164.657} C_VEL
LIN {X 0,Y 563.596,Z 704.89,A -85,B 0,C 180,E1 26163.275,E2 26163.275} C_VEL
LIN {X 0,Y 564.221,Z 684.63,A -85,B 0,C 180,E1 26162.107,E2 26162.107} C_VEL
LIN {X 0,Y 564.785,Z 664.484,A -85,B 0,C 180,E1 26161.158,E2 26161.158} C_VEL
LIN {X 0,Y 565.31,Z 642.965,A -85,B 0,C 180,E1 26160.345,E2 26160.345} C_VEL
LIN {X 0,Y 565.734,Z 621.321,A -85,B 0,C 180,E1 26159.734,E2 26159.734} C_VEL
LIN {X 0,Y 566.003,Z 601.115,A -85,B 0,C 180,E1 26159.336,E2 26159.336} C_VEL
LIN {X 0,Y 567.365,Z 375.938,A -85,B 0,C 180,E1 26156.104,E2 26156.104} C_VEL
LIN {X 0,Y 567.529,Z 316.819,A -85,B 0,C 180,E1 26155.228,E2 26155.228} C_VEL
LIN {X 0,Y 564.275,Z 305.623,A -85,B 0,C 180,E1 26154.806,E2 26154.806} C_VEL
LIN {X 0,Y 564.688,Z 284.044,A -85,B 0,C 180,E1 26152.323,E2 26152.323} C_VEL
LIN {X 0,Y 560.222,Z 270.569,A -85,B 0,C 180,E1 26150.284,E2 26150.284} C_VEL
LIN {X 0,Y 560.262,Z 270.437,A -85,B 0,C 180,E1 26147.162,E2 26147.162} C_VEL
LIN {X 0,Y 560.212,Z 270.436,A -85,B 0,C 180,E1 26144.112,E2 26144.112} C_VEL
LIN {X 0,Y 560.233,Z 270.446,A -85,B 0,C 180,E1 26140.784,E2 26140.784} C_VEL
LIN {X 0,Y 560.232,Z 270.433,A -85,B 0,C 180,E1 26137.746,E2 26137.746} C_VEL
LIN {X 0,Y 560.22,Z 270.445,A -85,B 0,C 180,E1 26134.456,E2 26134.456} C_VEL
LIN {X 0,Y 560.279,Z 270.445,A -85,B 0,C 180,E1 26131.264,E2 26131.264} C_VEL
LIN {X 0,Y 560.217,Z 270.447,A -85,B 0,C 180,E1 26128.111,E2 26128.111} C_VEL
LIN {X 0,Y 560.279,Z 270.443,A -85,B 0,C 180,E1 26124.908,E2 26124.908} C_VEL
LIN {X 0,Y 560.224,Z 270.446,A -85,B 0,C 180,E1 26121.791,E2 26121.791} C_VEL
LIN {X 0,Y 560.239,Z 270.444,A -85,B 0,C 180,E1 26118.415,E2 26118.415} C_VEL
LIN {X 0,Y 560.266,Z 270.44,A -85,B 0,C 180,E1 26115.209,E2 26115.209} C_VEL
LIN {X 0,Y 560.227,Z 270.445,A -85,B 0,C 180,E1 26111.948,E2 26111.948} C_VEL
LIN {X 0,Y 560.281,Z 270.438,A -85,B 0,C 180,E1 26108.725,E2 26108.725} C_VEL
LIN {X 0,Y 560.234,Z 270.447,A -85,B 0,C 180,E1 26105.53,E2 26105.53} C_VEL
LIN {X 0,Y 560.244,Z 270.438,A -85,B 0,C 180,E1 26102.148,E2 26102.148} C_VEL
LIN {X 0,Y 560.277,Z 270.448,A -85,B 0,C 180,E1 26098.977,E2 26098.977} C_VEL
LIN {X 0,Y 560.232,Z 270.439,A -85,B 0,C 180,E1 26095.701,E2 26095.701} C_VEL
LIN {X 0,Y 560.284,Z 270.439,A -85,B 0,C 180,E1 26092.412,E2 26092.412} C_VEL
LIN {X 0,Y 560.255,Z 270.441,A -85,B 0,C 180,E1 26089.096,E2 26089.096} C_VEL
LIN {X 0,Y 560.241,Z 270.441,A -85,B 0,C 180,E1 26085.711,E2 26085.711} C_VEL
LIN {X 0,Y 560.281,Z 270.444,A -85,B 0,C 180,E1 26082.447,E2 26082.447} C_VEL
LIN {X 0,Y 560.245,Z 270.446,A -85,B 0,C 180,E1 26079.197,E2 26079.197} C_VEL
LIN {X 0,Y 560.281,Z 270.442,A -85,B 0,C 180,E1 26076.242,E2 26076.242} C_VEL
LIN {X 0,Y 559.291,Z 270.563,A -85,B 0,C 180,E1 26075.454,E2 26075.454} C_VEL
LIN {X 0,Y 552.852,Z 271.373,A -85,B 0,C 180,E1 26073.243,E2 26073.243} C_VEL
LIN {X 0,Y 552.337,Z 271.437,A -85,B 0,C 180,E1 26072.667,E2 26072.667} C_VEL
LIN {X 0,Y 552.306,Z 271.434,A -85,B 0,C 180,E1 26069.302,E2 26069.302} C_VEL
LIN {X 0,Y 552.339,Z 271.43,A -85,B 0,C 180,E1 26065.989,E2 26065.989} C_VEL
LIN {X 0,Y 552.336,Z 271.436,A -85,B 0,C 180,E1 26062.624,E2 26062.624} C_VEL
LIN {X 0,Y 552.314,Z 271.432,A -85,B 0,C 180,E1 26059.329,E2 26059.329} C_VEL
LIN {X 0,Y 552.339,Z 271.433,A -85,B 0,C 180,E1 26056.092,E2 26056.092} C_VEL
LIN {X 0,Y 552.322,Z 271.436,A -85,B 0,C 180,E1 26052.753,E2 26052.753} C_VEL
LIN {X 0,Y 552.32,Z 271.431,A -85,B 0,C 180,E1 26049.315,E2 26049.315} C_VEL
LIN {X 0,Y 552.336,Z 271.433,A -85,B 0,C 180,E1 26045.985,E2 26045.985} C_VEL
LIN {X 0,Y 552.324,Z 271.435,A -85,B 0,C 180,E1 26042.646,E2 26042.646} C_VEL
LIN {X 0,Y 552.328,Z 271.429,A -85,B 0,C 180,E1 26039.245,E2 26039.245} C_VEL
LIN {X 0,Y 552.334,Z 271.432,A -85,B 0,C 180,E1 26035.883,E2 26035.883} C_VEL
LIN {X 0,Y 552.324,Z 271.435,A -85,B 0,C 180,E1 26032.567,E2 26032.567} C_VEL
LIN {X 0,Y 552.332,Z 271.43,A -85,B 0,C 180,E1 26029.126,E2 26029.126} C_VEL
LIN {X 0,Y 552.332,Z 271.434,A -85,B 0,C 180,E1 26025.755,E2 26025.755} C_VEL
LIN {X 0,Y 552.327,Z 271.436,A -85,B 0,C 180,E1 26022.44,E2 26022.44} C_VEL
LIN {X 0,Y 552.339,Z 271.429,A -85,B 0,C 180,E1 26019.061,E2 26019.061} C_VEL
LIN {X 0,Y 552.329,Z 271.434,A -85,B 0,C 180,E1 26015.714,E2 26015.714} C_VEL
LIN {X 0,Y 552.328,Z 271.434,A -85,B 0,C 180,E1 26012.386,E2 26012.386} C_VEL
LIN {X 0,Y 552.34,Z 271.428,A -85,B 0,C 180,E1 26008.963,E2 26008.963} C_VEL
LIN {X 0,Y 552.326,Z 271.434,A -85,B 0,C 180,E1 26005.536,E2 26005.536} C_VEL
LIN {X 0,Y 552.332,Z 271.435,A -85,B 0,C 180,E1 26002.197,E2 26002.197} C_VEL
LIN {X 0,Y 552.338,Z 271.429,A -85,B 0,C 180,E1 25998.832,E2 25998.832} C_VEL
LIN {X 0,Y 552.323,Z 271.435,A -85,B 0,C 180,E1 25995.427,E2 25995.427} C_VEL
LIN {X 0,Y 552.335,Z 271.435,A -85,B 0,C 180,E1 25992.077,E2 25992.077} C_VEL
LIN {X 0,Y 552.343,Z 271.428,A -85,B 0,C 180,E1 25988.664,E2 25988.664} C_VEL
LIN {X 0,Y 552.32,Z 271.433,A -85,B 0,C 180,E1 25985.281,E2 25985.281} C_VEL
LIN {X 0,Y 552.337,Z 271.434,A -85,B 0,C 180,E1 25981.924,E2 25981.924} C_VEL
LIN {X 0,Y 552.34,Z 271.428,A -85,B 0,C 180,E1 25978.497,E2 25978.497} C_VEL
LIN {X 0,Y 552.316,Z 271.434,A -85,B 0,C 180,E1 25975.091,E2 25975.091} C_VEL
LIN {X 0,Y 552.338,Z 271.436,A -85,B 0,C 180,E1 25971.751,E2 25971.751} C_VEL
LIN {X 0,Y 552.339,Z 271.429,A -85,B 0,C 180,E1 25968.369,E2 25968.369} C_VEL
LIN {X 0,Y 552.315,Z 271.435,A -85,B 0,C 180,E1 25965.058,E2 25965.058} C_VEL
LIN {X 0,Y 552.341,Z 271.434,A -85,B 0,C 180,E1 25961.771,E2 25961.771} C_VEL
LIN {X 0,Y 552.325,Z 271.431,A -85,B 0,C 180,E1 25958.388,E2 25958.388} C_VEL
LIN {X 0,Y 552.314,Z 271.436,A -85,B 0,C 180,E1 25955.02,E2 25955.02} C_VEL
LIN {X 0,Y 552.341,Z 271.434,A -85,B 0,C 180,E1 25951.666,E2 25951.666} C_VEL
LIN {X 0,Y 552.313,Z 271.432,A -85,B 0,C 180,E1 25948.383,E2 25948.383} C_VEL
LIN {X 0,Y 552.311,Z 271.436,A -85,B 0,C 180,E1 25944.914,E2 25944.914} C_VEL
LIN {X 0,Y 552.344,Z 271.432,A -85,B 0,C 180,E1 25941.671,E2 25941.671} C_VEL
LIN {X 0,Y 552.305,Z 271.433,A -85,B 0,C 180,E1 25938.361,E2 25938.361} C_VEL
LIN {X 0,Y 552.322,Z 271.43,A -85,B 0,C 180,E1 25935.003,E2 25935.003} C_VEL
LIN {X 0,Y 552.341,Z 271.431,A -85,B 0,C 180,E1 25931.678,E2 25931.678} C_VEL
LIN {X 0,Y 552.296,Z 271.431,A -85,B 0,C 180,E1 25928.327,E2 25928.327} C_VEL
LIN {X 0,Y 552.336,Z 271.431,A -85,B 0,C 180,E1 25925.089,E2 25925.089} C_VEL
LIN {X 0,Y 552.318,Z 271.428,A -85,B 0,C 180,E1 25921.764,E2 25921.764} C_VEL
LIN {X 0,Y 552.295,Z 271.429,A -85,B 0,C 180,E1 25918.444,E2 25918.444} C_VEL
LIN {X 0,Y 552.344,Z 271.429,A -85,B 0,C 180,E1 25915.223,E2 25915.223} C_VEL
LIN {X 0,Y 552.291,Z 271.428,A -85,B 0,C 180,E1 25911.987,E2 25911.987} C_VEL
LIN {X 0,Y 552.308,Z 271.437,A -85,B 0,C 180,E1 25908.619,E2 25908.619} C_VEL
LIN {X 0,Y 552.323,Z 271.427,A -85,B 0,C 180,E1 25905.426,E2 25905.426} C_VEL
LIN {X 0,Y 552.286,Z 271.436,A -85,B 0,C 180,E1 25902.184,E2 25902.184} C_VEL
LIN {X 0,Y 552.345,Z 271.425,A -85,B 0,C 180,E1 25898.997,E2 25898.997} C_VEL
LIN {X 0,Y 552.282,Z 271.434,A -85,B 0,C 180,E1 25895.842,E2 25895.842} C_VEL
LIN {X 0,Y 552.31,Z 271.438,A -85,B 0,C 180,E1 25892.503,E2 25892.503} C_VEL
LIN {X 0,Y 552.294,Z 271.43,A -85,B 0,C 180,E1 25889.422,E2 25889.422} C_VEL
LIN {X 0,Y 552.283,Z 271.435,A -85,B 0,C 180,E1 25886.11,E2 25886.11} C_VEL
LIN {X 0,Y 552.333,Z 271.428,A -85,B 0,C 180,E1 25882.929,E2 25882.929} C_VEL
LIN {X 0,Y 552.273,Z 271.436,A -85,B 0,C 180,E1 25879.735,E2 25879.735} C_VEL
LIN {X 0,Y 552.328,Z 271.417,A -85,B 0,C 180,E1 25876.536,E2 25876.536} C_VEL
LIN {X 0,Y 552.274,Z 271.44,A -85,B 0,C 180,E1 25873.449,E2 25873.449} C_VEL
LIN {X 0,Y 552.328,Z 271.624,A -85,B 0,C 180,E1 25870.24,E2 25870.24} C_VEL
LIN {X 0,Y 557.632,Z 287.637,A -85,B 0,C 180,E1 25867.802,E2 25867.802} C_VEL
LIN {X 0,Y 557.123,Z 305.792,A -85,B 0,C 180,E1 25865.704,E2 25865.704} C_VEL
LIN {X 0,Y 561.132,Z 320.122,A -85,B 0,C 180,E1 25865.176,E2 25865.176} C_VEL
LIN {X 0,Y 559.562,Z 539.79,A -85,B 0,C 180,E1 25861.972,E2 25861.972} C_VEL
LIN {X 0,Y 559.042,Z 608.396,A -85,B 0,C 180,E1 25860.958,E2 25860.958} C_VEL
LIN {X 0,Y 558.578,Z 631.697,A -85,B 0,C 180,E1 25860.412,E2 25860.412} C_VEL
LIN {X 0,Y 558.029,Z 653.488,A -85,B 0,C 180,E1 25859.691,E2 25859.691} C_VEL
LIN {X 0,Y 557.352,Z 675.643,A -85,B 0,C 180,E1 25858.735,E2 25858.735} C_VEL
LIN {X 0,Y 556.698,Z 693.719,A -85,B 0,C 180,E1 25857.779,E2 25857.779} C_VEL
LIN {X 0,Y 555.957,Z 714.195,A -85,B 0,C 180,E1 25856.487,E2 25856.487} C_VEL
LIN {X 0,Y 555.195,Z 733.16,A -85,B 0,C 180,E1 25855.061,E2 25855.061} C_VEL
LIN {X 0,Y 554.503,Z 751.11,A -85,B 0,C 180,E1 25853.484,E2 25853.484} C_VEL
LIN {X 0,Y 553.85,Z 768.208,A -85,B 0,C 180,E1 25851.72,E2 25851.72} C_VEL
LIN {X 0,Y 553.295,Z 783.749,A -85,B 0,C 180,E1 25849.86,E2 25849.86} C_VEL
LIN {X 0,Y 552.85,Z 797.732,A -85,B 0,C 180,E1 25847.905,E2 25847.905} C_VEL
LIN {X 0,Y 552.512,Z 809.721,A -85,B 0,C 180,E1 25845.966,E2 25845.966} C_VEL
LIN {X 0,Y 552.244,Z 821.392,A -85,B 0,C 180,E1 25843.72,E2 25843.72} C_VEL
LIN {X 0,Y 552.081,Z 830.712,A -85,B 0,C 180,E1 25841.54,E2 25841.54} C_VEL
LIN {X 0,Y 551.99,Z 838.539,A -85,B 0,C 180,E1 25839.277,E2 25839.277} C_VEL
LIN {X 0,Y 551.942,Z 844.165,A -85,B 0,C 180,E1 25837.18,E2 25837.18} C_VEL
LIN {X 0,Y 551.919,Z 848.652,A -85,B 0,C 180,E1 25834.878,E2 25834.878} C_VEL
LIN {X 0,Y 551.907,Z 851.393,A -85,B 0,C 180,E1 25832.596,E2 25832.596} C_VEL
LIN {X 0,Y 551.898,Z 852.417,A -85,B 0,C 180,E1 25830.415,E2 25830.415} C_VEL
LIN {X 0,Y 551.907,Z 851.894,A -85,B 0,C 180,E1 25828.131,E2 25828.131} C_VEL
LIN {X 0,Y 551.913,Z 849.849,A -85,B 0,C 180,E1 25825.949,E2 25825.949} C_VEL
LIN {X 0,Y 551.921,Z 846.209,A -85,B 0,C 180,E1 25823.76,E2 25823.76} C_VEL
LIN {X 0,Y 551.951,Z 840.665,A -85,B 0,C 180,E1 25821.458,E2 25821.458} C_VEL
LIN {X 0,Y 552.027,Z 834.397,A -85,B 0,C 180,E1 25819.459,E2 25819.459} C_VEL
LIN {X 0,Y 552.157,Z 825.7,A -85,B 0,C 180,E1 25817.237,E2 25817.237} C_VEL
LIN {X 0,Y 552.364,Z 815.542,A -85,B 0,C 180,E1 25815.106,E2 25815.106} C_VEL
LIN {X 0,Y 552.666,Z 803.986,A -85,B 0,C 180,E1 25813.066,E2 25813.066} C_VEL
LIN {X 0,Y 553.082,Z 790.246,A -85,B 0,C 180,E1 25811.011,E2 25811.011} C_VEL
LIN {X 0,Y 553.611,Z 774.916,A -85,B 0,C 180,E1 25809.048,E2 25809.048} C_VEL
LIN {X 0,Y 554.198,Z 758.881,A -85,B 0,C 180,E1 25807.289,E2 25807.289} C_VEL
LIN {X 0,Y 554.82,Z 742.614,A -85,B 0,C 180,E1 25805.74,E2 25805.74} C_VEL
LIN {X 0,Y 555.593,Z 723.529,A -85,B 0,C 180,E1 25804.183,E2 25804.183} C_VEL
LIN {X 0,Y 556.341,Z 704.005,A -85,B 0,C 180,E1 25802.84,E2 25802.84} C_VEL
LIN {X 0,Y 557.089,Z 682.392,A -85,B 0,C 180,E1 25801.601,E2 25801.601} C_VEL
LIN {X 0,Y 557.738,Z 663.156,A -85,B 0,C 180,E1 25800.699,E2 25800.699} C_VEL
LIN {X 0,Y 558.346,Z 641.582,A -85,B 0,C 180,E1 25799.889,E2 25799.889} C_VEL
LIN {X 0,Y 558.819,Z 620.231,A -85,B 0,C 180,E1 25799.293,E2 25799.293} C_VEL
LIN {X 0,Y 559.136,Z 599.756,A -85,B 0,C 180,E1 25798.894,E2 25798.894} C_VEL
LIN {X 0,Y 560.721,Z 376.339,A -85,B 0,C 180,E1 25795.653,E2 25795.653} C_VEL
LIN {X 0,Y 560.967,Z 318.827,A -85,B 0,C 180,E1 25794.792,E2 25794.792} C_VEL
LIN {X 0,Y 557.1,Z 305.646,A -85,B 0,C 180,E1 25794.287,E2 25794.287} C_VEL
LIN {X 0,Y 557.575,Z 287.475,A -85,B 0,C 180,E1 25792.174,E2 25792.174} C_VEL
LIN {X 0,Y 552.855,Z 273.585,A -85,B 0,C 180,E1 25790.069,E2 25790.069} C_VEL
LIN {X 0,Y 552.315,Z 271.49,A -85,B 0,C 180,E1 25789.703,E2 25789.703} C_VEL
LIN {X 0,Y 552.273,Z 271.44,A -85,B 0,C 180,E1 25786.532,E2 25786.532} C_VEL
LIN {X 0,Y 552.337,Z 271.418,A -85,B 0,C 180,E1 25783.307,E2 25783.307} C_VEL
LIN {X 0,Y 552.274,Z 271.437,A -85,B 0,C 180,E1 25780.129,E2 25780.129} C_VEL
LIN {X 0,Y 552.305,Z 271.435,A -85,B 0,C 180,E1 25776.814,E2 25776.814} C_VEL
LIN {X 0,Y 552.303,Z 271.434,A -85,B 0,C 180,E1 25773.619,E2 25773.619} C_VEL
LIN {X 0,Y 552.28,Z 271.43,A -85,B 0,C 180,E1 25770.283,E2 25770.283} C_VEL
LIN {X 0,Y 552.345,Z 271.428,A -85,B 0,C 180,E1 25767.052,E2 25767.052} C_VEL
LIN {X 0,Y 552.286,Z 271.435,A -85,B 0,C 180,E1 25763.811,E2 25763.811} C_VEL
LIN {X 0,Y 552.3,Z 271.425,A -85,B 0,C 180,E1 25760.45,E2 25760.45} C_VEL
LIN {X 0,Y 552.325,Z 271.437,A -85,B 0,C 180,E1 25757.271,E2 25757.271} C_VEL
LIN {X 0,Y 552.286,Z 271.428,A -85,B 0,C 180,E1 25753.988,E2 25753.988} C_VEL
LIN {X 0,Y 552.342,Z 271.427,A -85,B 0,C 180,E1 25750.746,E2 25750.746} C_VEL
LIN {X 0,Y 552.299,Z 271.431,A -85,B 0,C 180,E1 25747.49,E2 25747.49} C_VEL
LIN {X 0,Y 552.296,Z 271.429,A -85,B 0,C 180,E1 25744.049,E2 25744.049} C_VEL
LIN {X 0,Y 552.344,Z 271.434,A -85,B 0,C 180,E1 25740.83,E2 25740.83} C_VEL
LIN {X 0,Y 552.295,Z 271.431,A -85,B 0,C 180,E1 25737.614,E2 25737.614} C_VEL
LIN {X 0,Y 552.33,Z 271.431,A -85,B 0,C 180,E1 25734.286,E2 25734.286} C_VEL
LIN {X 0,Y 552.331,Z 271.428,A -85,B 0,C 180,E1 25730.939,E2 25730.939} C_VEL
LIN {X 0,Y 552.298,Z 271.434,A -85,B 0,C 180,E1 25727.665,E2 25727.665} C_VEL
LIN {X 0,Y 552.344,Z 271.425,A -85,B 0,C 180,E1 25724.352,E2 25724.352} C_VEL
LIN {X 0,Y 552.321,Z 271.437,A -85,B 0,C 180,E1 25720.983,E2 25720.983} C_VEL
LIN {X 0,Y 552.308,Z 271.433,A -85,B 0,C 180,E1 25717.656,E2 25717.656} C_VEL
LIN {X 0,Y 552.342,Z 271.433,A -85,B 0,C 180,E1 25714.351,E2 25714.351} C_VEL
LIN {X 0,Y 552.337,Z 271.437,A -85,B 0,C 180,E1 25712.667,E2 25712.667} C_VEL
LIN {X 0,Y 551.361,Z 271.559,A -85,B 0,C 180,E1 25711.868,E2 25711.868} C_VEL
LIN {X 0,Y 544.894,Z 272.357,A -85,B 0,C 180,E1 25709.624,E2 25709.624} C_VEL
LIN {X 0,Y 544.374,Z 272.425,A -85,B 0,C 180,E1 25709.04,E2 25709.04} C_VEL
LIN {X 0,Y 544.377,Z 272.421,A -85,B 0,C 180,E1 25705.549,E2 25705.549} C_VEL
LIN {X 0,Y 544.402,Z 272.424,A -85,B 0,C 180,E1 25702.295,E2 25702.295} C_VEL
LIN {X 0,Y 544.375,Z 272.424,A -85,B 0,C 180,E1 25699.014,E2 25699.014} C_VEL
LIN {X 0,Y 544.391,Z 272.419,A -85,B 0,C 180,E1 25695.592,E2 25695.592} C_VEL
LIN {X 0,Y 544.401,Z 272.425,A -85,B 0,C 180,E1 25692.236,E2 25692.236} C_VEL
LIN {X 0,Y 544.376,Z 272.424,A -85,B 0,C 180,E1 25688.913,E2 25688.913} C_VEL
LIN {X 0,Y 544.396,Z 272.418,A -85,B 0,C 180,E1 25685.476,E2 25685.476} C_VEL
LIN {X 0,Y 544.398,Z 272.423,A -85,B 0,C 180,E1 25682.058,E2 25682.058} C_VEL
LIN {X 0,Y 544.38,Z 272.422,A -85,B 0,C 180,E1 25678.764,E2 25678.764} C_VEL
LIN {X 0,Y 544.397,Z 272.417,A -85,B 0,C 180,E1 25675.336,E2 25675.336} C_VEL
LIN {X 0,Y 544.397,Z 272.423,A -85,B 0,C 180,E1 25671.952,E2 25671.952} C_VEL
LIN {X 0,Y 544.384,Z 272.424,A -85,B 0,C 180,E1 25668.608,E2 25668.608} C_VEL
LIN {X 0,Y 544.404,Z 272.418,A -85,B 0,C 180,E1 25665.226,E2 25665.226} C_VEL
LIN {X 0,Y 544.393,Z 272.424,A -85,B 0,C 180,E1 25661.782,E2 25661.782} C_VEL
LIN {X 0,Y 544.388,Z 272.424,A -85,B 0,C 180,E1 25658.449,E2 25658.449} C_VEL
LIN {X 0,Y 544.4,Z 272.418,A -85,B 0,C 180,E1 25655.058,E2 25655.058} C_VEL
LIN {X 0,Y 544.392,Z 272.422,A -85,B 0,C 180,E1 25651.684,E2 25651.684} C_VEL
LIN {X 0,Y 544.392,Z 272.423,A -85,B 0,C 180,E1 25648.316,E2 25648.316} C_VEL
LIN {X 0,Y 544.399,Z 272.418,A -85,B 0,C 180,E1 25644.837,E2 25644.837} C_VEL
LIN {X 0,Y 544.386,Z 272.423,A -85,B 0,C 180,E1 25641.445,E2 25641.445} C_VEL
LIN {X 0,Y 544.399,Z 272.425,A -85,B 0,C 180,E1 25638.022,E2 25638.022} C_VEL
LIN {X 0,Y 544.399,Z 272.419,A -85,B 0,C 180,E1 25634.556,E2 25634.556} C_VEL
LIN {X 0,Y 544.383,Z 272.421,A -85,B 0,C 180,E1 25631.141,E2 25631.141} C_VEL
LIN {X 0,Y 544.407,Z 272.425,A -85,B 0,C 180,E1 25627.766,E2 25627.766} C_VEL
LIN {X 0,Y 544.398,Z 272.419,A -85,B 0,C 180,E1 25624.314,E2 25624.314} C_VEL
LIN {X 0,Y 544.382,Z 272.42,A -85,B 0,C 180,E1 25620.957,E2 25620.957} C_VEL
LIN {X 0,Y 544.396,Z 272.425,A -85,B 0,C 180,E1 25617.569,E2 25617.569} C_VEL
LIN {X 0,Y 544.398,Z 272.42,A -85,B 0,C 180,E1 25614.136,E2 25614.136} C_VEL
LIN {X 0,Y 544.378,Z 272.421,A -85,B 0,C 180,E1 25610.813,E2 25610.813} C_VEL
LIN {X 0,Y 544.395,Z 272.425,A -85,B 0,C 180,E1 25607.433,E2 25607.433} C_VEL
LIN {X 0,Y 544.404,Z 272.42,A -85,B 0,C 180,E1 25604.103,E2 25604.103} C_VEL
LIN {X 0,Y 544.372,Z 272.423,A -85,B 0,C 180,E1 25600.825,E2 25600.825} C_VEL
LIN {X 0,Y 544.403,Z 272.424,A -85,B 0,C 180,E1 25597.496,E2 25597.496} C_VEL
LIN {X 0,Y 544.399,Z 272.419,A -85,B 0,C 180,E1 25594.068,E2 25594.068} C_VEL
LIN {X 0,Y 544.368,Z 272.423,A -85,B 0,C 180,E1 25590.704,E2 25590.704} C_VEL
LIN {X 0,Y 544.398,Z 272.427,A -85,B 0,C 180,E1 25587.333,E2 25587.333} C_VEL
LIN {X 0,Y 544.397,Z 272.419,A -85,B 0,C 180,E1 25583.947,E2 25583.947} C_VEL
LIN {X 0,Y 544.364,Z 272.423,A -85,B 0,C 180,E1 25580.65,E2 25580.65} C_VEL
LIN {X 0,Y 544.402,Z 272.422,A -85,B 0,C 180,E1 25577.309,E2 25577.309} C_VEL
LIN {X 0,Y 544.385,Z 272.416,A -85,B 0,C 180,E1 25573.922,E2 25573.922} C_VEL
LIN {X 0,Y 544.361,Z 272.415,A -85,B 0,C 180,E1 25570.584,E2 25570.584} C_VEL
LIN {X 0,Y 544.406,Z 272.421,A -85,B 0,C 180,E1 25567.28,E2 25567.28} C_VEL
LIN {X 0,Y 544.365,Z 272.413,A -85,B 0,C 180,E1 25564.002,E2 25564.002} C_VEL
LIN {X 0,Y 544.359,Z 272.425,A -85,B 0,C 180,E1 25560.526,E2 25560.526} C_VEL
LIN {X 0,Y 544.404,Z 272.412,A -85,B 0,C 180,E1 25557.263,E2 25557.263} C_VEL
LIN {X 0,Y 544.355,Z 272.423,A -85,B 0,C 180,E1 25553.99,E2 25553.99} C_VEL
LIN {X 0,Y 544.366,Z 272.419,A -85,B 0,C 180,E1 25550.592,E2 25550.592} C_VEL
LIN {X 0,Y 544.391,Z 272.422,A -85,B 0,C 180,E1 25547.375,E2 25547.375} C_VEL
LIN {X 0,Y 544.347,Z 272.42,A -85,B 0,C 180,E1 25544.116,E2 25544.116} C_VEL
LIN {X 0,Y 544.395,Z 272.419,A -85,B 0,C 180,E1 25540.807,E2 25540.807} C_VEL
LIN {X 0,Y 544.351,Z 272.422,A -85,B 0,C 180,E1 25537.653,E2 25537.653} C_VEL
LIN {X 0,Y 544.347,Z 272.418,A -85,B 0,C 180,E1 25534.194,E2 25534.194} C_VEL
LIN {X 0,Y 544.406,Z 272.424,A -85,B 0,C 180,E1 25530.95,E2 25530.95} C_VEL
LIN {X 0,Y 544.341,Z 272.426,A -85,B 0,C 180,E1 25527.663,E2 25527.663} C_VEL
LIN {X 0,Y 544.355,Z 272.426,A -85,B 0,C 180,E1 25524.261,E2 25524.261} C_VEL
LIN {X 0,Y 544.37,Z 272.401,A -85,B 0,C 180,E1 25521.086,E2 25521.086} C_VEL
LIN {X 0,Y 544.336,Z 272.425,A -85,B 0,C 180,E1 25517.899,E2 25517.899} C_VEL
LIN {X 0,Y 544.399,Z 272.415,A -85,B 0,C 180,E1 25514.701,E2 25514.701} C_VEL
LIN {X 0,Y 544.329,Z 272.405,A -85,B 0,C 180,E1 25511.458,E2 25511.458} C_VEL
LIN {X 0,Y 544.424,Z 272.65,A -85,B 0,C 180,E1 25510.761,E2 25510.761} C_VEL
LIN {X 0,Y 550.398,Z 290.694,A -85,B 0,C 180,E1 25508.011,E2 25508.011} C_VEL
LIN {X 0,Y 550.021,Z 305.934,A -85,B 0,C 180,E1 25506.233,E2 25506.233} C_VEL
LIN {X 0,Y 554.575,Z 322.094,A -85,B 0,C 180,E1 25505.624,E2 25505.624} C_VEL
LIN {X 0,Y 552.767,Z 541.063,A -85,B 0,C 180,E1 25502.394,E2 25502.394} C_VEL
LIN {X 0,Y 552.176,Z 608.374,A -85,B 0,C 180,E1 25501.386,E2 25501.386} C_VEL
LIN {X 0,Y 551.642,Z 631.54,A -85,B 0,C 180,E1 25500.84,E2 25500.84} C_VEL
LIN {X 0,Y 551.053,Z 652.549,A -85,B 0,C 180,E1 25500.141,E2 25500.141} C_VEL
LIN {X 0,Y 550.326,Z 673.38,A -85,B 0,C 180,E1 25499.256,E2 25499.256} C_VEL
LIN {X 0,Y 549.534,Z 692.73,A -85,B 0,C 180,E1 25498.232,E2 25498.232} C_VEL
LIN {X 0,Y 548.707,Z 712.444,A -85,B 0,C 180,E1 25496.994,E2 25496.994} C_VEL
LIN {X 0,Y 547.837,Z 731.39,A -85,B 0,C 180,E1 25495.571,E2 25495.571} C_VEL
LIN {X 0,Y 547.079,Z 748.093,A -85,B 0,C 180,E1 25494.108,E2 25494.108} C_VEL
LIN {X 0,Y 546.273,Z 766.215,A -85,B 0,C 180,E1 25492.264,E2 25492.264} C_VEL
LIN {X 0,Y 545.608,Z 782.053,A -85,B 0,C 180,E1 25490.376,E2 25490.376} C_VEL
LIN {X 0,Y 545.065,Z 796.311,A -85,B 0,C 180,E1 25488.391,E2 25488.391} C_VEL
LIN {X 0,Y 544.684,Z 807.822,A -85,B 0,C 180,E1 25486.53,E2 25486.53} C_VEL
LIN {X 0,Y 544.36,Z 819.32,A -85,B 0,C 180,E1 25484.357,E2 25484.357} C_VEL
LIN {X 0,Y 544.145,Z 828.948,A -85,B 0,C 180,E1 25482.167,E2 25482.167} C_VEL
LIN {X 0,Y 544.022,Z 836.537,A -85,B 0,C 180,E1 25480.055,E2 25480.055} C_VEL
LIN {X 0,Y 543.95,Z 843.152,A -85,B 0,C 180,E1 25477.711,E2 25477.711} C_VEL
LIN {X 0,Y 543.925,Z 847.606,A -85,B 0,C 180,E1 25475.591,E2 25475.591} C_VEL
LIN {X 0,Y 543.914,Z 850.694,A -85,B 0,C 180,E1 25473.372,E2 25473.372} C_VEL
LIN {X 0,Y 543.914,Z 852.276,A -85,B 0,C 180,E1 25471.053,E2 25471.053} C_VEL
LIN {X 0,Y 543.914,Z 852.276,A -85,B 0,C 180,E1 25468.947,E2 25468.947} C_VEL
LIN {X 0,Y 543.914,Z 850.694,A -85,B 0,C 180,E1 25466.628,E2 25466.628} C_VEL
LIN {X 0,Y 543.925,Z 847.606,A -85,B 0,C 180,E1 25464.409,E2 25464.409} C_VEL
LIN {X 0,Y 543.95,Z 843.152,A -85,B 0,C 180,E1 25462.289,E2 25462.289} C_VEL
LIN {X 0,Y 544.022,Z 836.537,A -85,B 0,C 180,E1 25459.945,E2 25459.945} C_VEL
LIN {X 0,Y 544.148,Z 828.82,A -85,B 0,C 180,E1 25457.801,E2 25457.801} C_VEL
LIN {X 0,Y 544.36,Z 819.32,A -85,B 0,C 180,E1 25455.643,E2 25455.643} C_VEL
LIN {X 0,Y 544.684,Z 807.822,A -85,B 0,C 180,E1 25453.47,E2 25453.47} C_VEL
LIN {X 0,Y 545.094,Z 795.602,A -85,B 0,C 180,E1 25451.499,E2 25451.499} C_VEL
LIN {X 0,Y 545.659,Z 780.664,A -85,B 0,C 180,E1 25449.447,E2 25449.447} C_VEL
